LIN {X 0,Y 474.72,Z 465.35,A -85,B 0,C 180,E1 -7388.514,E2 -7388.514} C_VEL
LIN {X 0,Y 474.696,Z 465.35,A -85,B 0,C 180,E1 -7391.963,E2 -7391.963} C_VEL
LIN {X 0,Y 474.691,Z 465.345,A -85,B 0,C 180,E1 -7395.456,E2 -7395.456} C_VEL
LIN {X 0,Y 474.657,Z 465.36,A -85,B 0,C 180,E1 -7399.011,E2 -7399.011} C_VEL
LIN {X 0,Y 474.581,Z 465.36,A -85,B 0,C 180,E1 -7401.729,E2 -7401.729} C_VEL
LIN {X 0,Y 474.651,Z 465.358,A -85,B 0,C 180,E1 -7404.493,E2 -7404.493} C_VEL
LIN {X 0,Y 474.692,Z 465.348,A -85,B 0,C 180,E1 -7407.339,E2 -7407.339} C_VEL
LIN {X 0,Y 474.603,Z 465.346,A -85,B 0,C 180,E1 -7410.812,E2 -7410.812} C_VEL
LIN {X 0,Y 474.632,Z 465.355,A -85,B 0,C 180,E1 -7413.985,E2 -7413.985} C_VEL
LIN {X 0,Y 474.57,Z 465.371,A -85,B 0,C 180,E1 -7416.901,E2 -7416.901} C_VEL
LIN {X 0,Y 474.613,Z 465.345,A -85,B 0,C 180,E1 -7419.647,E2 -7419.647} C_VEL
LIN {X 0,Y 474.627,Z 465.363,A -85,B 0,C 180,E1 -7422.933,E2 -7422.933} C_VEL
LIN {X 0,Y 474.611,Z 465.357,A -85,B 0,C 180,E1 -7425.897,E2 -7425.897} C_VEL
LIN {X 0,Y 474.629,Z 465.361,A -85,B 0,C 180,E1 -7429.041,E2 -7429.041} C_VEL
LIN {X 0,Y 474.613,Z 465.359,A -85,B 0,C 180,E1 -7431.704,E2 -7431.704} C_VEL
LIN {X 0,Y 474.627,Z 465.337,A -85,B 0,C 180,E1 -7434.727,E2 -7434.727} C_VEL
LIN {X 0,Y 474.637,Z 465.356,A -85,B 0,C 180,E1 -7437.789,E2 -7437.789} C_VEL
LIN {X 0,Y 474.624,Z 465.363,A -85,B 0,C 180,E1 -7440.885,E2 -7440.885} C_VEL
LIN {X 0,Y 474.661,Z 465.347,A -85,B 0,C 180,E1 -7443.629,E2 -7443.629} C_VEL
LIN {X 0,Y 474.637,Z 465.361,A -85,B 0,C 180,E1 -7446.642,E2 -7446.642} C_VEL
LIN {X 0,Y 474.659,Z 465.358,A -85,B 0,C 180,E1 -7450.09,E2 -7450.09} C_VEL
LIN {X 0,Y 474.656,Z 465.329,A -85,B 0,C 180,E1 -7451.688,E2 -7451.688} C_VEL
LIN {X 0,Y 474.507,Z 466.016,A -85,B 0,C 180,E1 -7452.131,E2 -7452.131} C_VEL
LIN {X 0,Y 474.153,Z 467.747,A -85,B 0,C 180,E1 -7452.533,E2 -7452.533} C_VEL
LIN {X 0,Y 473.419,Z 471.634,A -85,B 0,C 180,E1 -7453.047,E2 -7453.047} C_VEL
LIN {X 0,Y 472.593,Z 476.648,A -85,B 0,C 180,E1 -7453.451,E2 -7453.451} C_VEL
LIN {X 0,Y 471.86,Z 482.314,A -85,B 0,C 180,E1 -7453.745,E2 -7453.745} C_VEL
LIN {X 0,Y 471.447,Z 488.35,A -85,B 0,C 180,E1 -7453.907,E2 -7453.907} C_VEL
LIN {X 0,Y 471.092,Z 547.467,A -85,B 0,C 180,E1 -7454.839,E2 -7454.839} C_VEL
LIN {X 0,Y 471.01,Z 560.516,A -85,B 0,C 180,E1 -7455.223,E2 -7455.223} C_VEL
LIN {X 0,Y 470.78,Z 572.512,A -85,B 0,C 180,E1 -7455.741,E2 -7455.741} C_VEL
LIN {X 0,Y 470.513,Z 583.759,A -85,B 0,C 180,E1 -7456.392,E2 -7456.392} C_VEL
LIN {X 0,Y 470.007,Z 595.351,A -85,B 0,C 180,E1 -7457.259,E2 -7457.259} C_VEL
LIN {X 0,Y 469.554,Z 605.694,A -85,B 0,C 180,E1 -7458.233,E2 -7458.233} C_VEL
LIN {X 0,Y 469.147,Z 614.13,A -85,B 0,C 180,E1 -7459.208,E2 -7459.208} C_VEL
LIN {X 0,Y 468.818,Z 621.878,A -85,B 0,C 180,E1 -7460.291,E2 -7460.291} C_VEL
LIN {X 0,Y 468.374,Z 629.568,A -85,B 0,C 180,E1 -7461.609,E2 -7461.609} C_VEL
LIN {X 0,Y 468.091,Z 635.326,A -85,B 0,C 180,E1 -7462.84,E2 -7462.84} C_VEL
LIN {X 0,Y 467.937,Z 639.602,A -85,B 0,C 180,E1 -7463.965,E2 -7463.965} C_VEL
LIN {X 0,Y 467.644,Z 643.493,A -85,B 0,C 180,E1 -7465.259,E2 -7465.259} C_VEL
LIN {X 0,Y 467.456,Z 646.362,A -85,B 0,C 180,E1 -7466.552,E2 -7466.552} C_VEL
LIN {X 0,Y 467.483,Z 647.723,A -85,B 0,C 180,E1 -7467.415,E2 -7467.415} C_VEL
LIN {X 0,Y 467.356,Z 648.71,A -85,B 0,C 180,E1 -7468.277,E2 -7468.277} C_VEL
LIN {X 0,Y 467.432,Z 649.296,A -85,B 0,C 180,E1 -7469.139,E2 -7469.139} C_VEL
LIN {X 0,Y 467.416,Z 649.528,A -85,B 0,C 180,E1 -7470,E2 -7470} C_VEL
LIN {X 0,Y 467.432,Z 649.346,A -85,B 0,C 180,E1 -7470.861,E2 -7470.861} C_VEL
LIN {X 0,Y 467.356,Z 648.79,A -85,B 0,C 180,E1 -7471.723,E2 -7471.723} C_VEL
LIN {X 0,Y 467.482,Z 647.836,A -85,B 0,C 180,E1 -7472.585,E2 -7472.585} C_VEL
LIN {X 0,Y 467.451,Z 646.526,A -85,B 0,C 180,E1 -7473.448,E2 -7473.448} C_VEL
LIN {X 0,Y 467.639,Z 643.718,A -85,B 0,C 180,E1 -7474.741,E2 -7474.741} C_VEL
LIN {X 0,Y 467.925,Z 639.903,A -85,B 0,C 180,E1 -7476.035,E2 -7476.035} C_VEL
LIN {X 0,Y 468.063,Z 634.827,A -85,B 0,C 180,E1 -7477.377,E2 -7477.377} C_VEL
LIN {X 0,Y 468.404,Z 628.813,A -85,B 0,C 180,E1 -7478.629,E2 -7478.629} C_VEL
LIN {X 0,Y 468.879,Z 621.039,A -85,B 0,C 180,E1 -7479.926,E2 -7479.926} C_VEL
LIN {X 0,Y 469.297,Z 611.375,A -85,B 0,C 180,E1 -7481.226,E2 -7481.226} C_VEL
LIN {X 0,Y 469.741,Z 602.348,A -85,B 0,C 180,E1 -7482.2,E2 -7482.2} C_VEL
LIN {X 0,Y 470.229,Z 591.863,A -85,B 0,C 180,E1 -7483.114,E2 -7483.114} C_VEL
LIN {X 0,Y 470.571,Z 580.37,A -85,B 0,C 180,E1 -7483.914,E2 -7483.914} C_VEL
LIN {X 0,Y 470.851,Z 569.136,A -85,B 0,C 180,E1 -7484.517,E2 -7484.517} C_VEL
LIN {X 0,Y 471.03,Z 555.98,A -85,B 0,C 180,E1 -7485.025,E2 -7485.025} C_VEL
LIN {X 0,Y 471.055,Z 542.285,A -85,B 0,C 180,E1 -7485.356,E2 -7485.356} C_VEL
LIN {X 0,Y 471.382,Z 476.884,A -85,B 0,C 180,E1 -7486.367,E2 -7486.367} C_VEL
LIN {X 0,Y 467.762,Z 467.093,A -85,B 0,C 180,E1 -7486.689,E2 -7486.689} C_VEL
LIN {X 0,Y 467.626,Z 466.313,A -85,B 0,C 180,E1 -7486.855,E2 -7486.855} C_VEL
LIN {X 0,Y 467.626,Z 466.222,A -85,B 0,C 180,E1 -7489.307,E2 -7489.307} C_VEL
LIN {X 0,Y 467.535,Z 466.233,A -85,B 0,C 180,E1 -7492.073,E2 -7492.073} C_VEL
LIN {X 0,Y 467.604,Z 466.24,A -85,B 0,C 180,E1 -7494.887,E2 -7494.887} C_VEL
LIN {X 0,Y 467.62,Z 466.22,A -85,B 0,C 180,E1 -7497.768,E2 -7497.768} C_VEL
LIN {X 0,Y 467.569,Z 466.243,A -85,B 0,C 180,E1 -7501.044,E2 -7501.044} C_VEL
LIN {X 0,Y 467.588,Z 466.237,A -85,B 0,C 180,E1 -7504.242,E2 -7504.242} C_VEL
LIN {X 0,Y 467.548,Z 466.24,A -85,B 0,C 180,E1 -7507.186,E2 -7507.186} C_VEL
LIN {X 0,Y 467.576,Z 466.239,A -85,B 0,C 180,E1 -7510.264,E2 -7510.264} C_VEL
LIN {X 0,Y 467.583,Z 466.231,A -85,B 0,C 180,E1 -7512.566,E2 -7512.566} C_VEL
LIN {X 0,Y 467.567,Z 466.243,A -85,B 0,C 180,E1 -7515.052,E2 -7515.052} C_VEL
LIN {X 0,Y 467.584,Z 466.237,A -85,B 0,C 180,E1 -7517.439,E2 -7517.439} C_VEL
LIN {X 0,Y 467.555,Z 466.226,A -85,B 0,C 180,E1 -7520.852,E2 -7520.852} C_VEL
LIN {X 0,Y 467.557,Z 466.24,A -85,B 0,C 180,E1 -7524.259,E2 -7524.259} C_VEL
LIN {X 0,Y 467.576,Z 466.229,A -85,B 0,C 180,E1 -7527.32,E2 -7527.32} C_VEL
LIN {X 0,Y 467.571,Z 466.222,A -85,B 0,C 180,E1 -7530.665,E2 -7530.665} C_VEL
LIN {X 0,Y 467.621,Z 466.235,A -85,B 0,C 180,E1 -7533.2,E2 -7533.2} C_VEL
LIN {X 0,Y 467.585,Z 466.234,A -85,B 0,C 180,E1 -7536.468,E2 -7536.468} C_VEL
LIN {X 0,Y 467.615,Z 466.235,A -85,B 0,C 180,E1 -7539.777,E2 -7539.777} C_VEL
LIN {X 0,Y 467.6,Z 466.232,A -85,B 0,C 180,E1 -7542.506,E2 -7542.506} C_VEL
LIN {X 0,Y 467.6,Z 466.235,A -85,B 0,C 180,E1 -7545.196,E2 -7545.196} C_VEL
LIN {X 0,Y 467.647,Z 466.229,A -85,B 0,C 180,E1 -7547.854,E2 -7547.854} C_VEL
LIN {X 0,Y 467.673,Z 466.224,A -85,B 0,C 180,E1 -7551.357,E2 -7551.357} C_VEL
LIN {X 0,Y 467.735,Z 466.218,A -85,B 0,C 180,E1 -7553.962,E2 -7553.962} C_VEL
LIN {X 0,Y 467.851,Z 466.2,A -85,B 0,C 180,E1 -7557.417,E2 -7557.417} C_VEL
LIN {X 0,Y 467.873,Z 466.201,A -85,B 0,C 180,E1 -7560,E2 -7560} C_VEL
LIN {X 0,Y 467.851,Z 466.199,A -85,B 0,C 180,E1 -7562.583,E2 -7562.583} C_VEL
LIN {X 0,Y 467.742,Z 466.217,A -85,B 0,C 180,E1 -7566.037,E2 -7566.037} C_VEL
LIN {X 0,Y 467.673,Z 466.224,A -85,B 0,C 180,E1 -7568.643,E2 -7568.643} C_VEL
LIN {X 0,Y 467.647,Z 466.227,A -85,B 0,C 180,E1 -7572.146,E2 -7572.146} C_VEL
LIN {X 0,Y 467.63,Z 466.233,A -85,B 0,C 180,E1 -7575.695,E2 -7575.695} C_VEL
LIN {X 0,Y 467.608,Z 466.219,A -85,B 0,C 180,E1 -7578.765,E2 -7578.765} C_VEL
LIN {X 0,Y 467.571,Z 466.236,A -85,B 0,C 180,E1 -7581.269,E2 -7581.269} C_VEL
LIN {X 0,Y 467.565,Z 466.241,A -85,B 0,C 180,E1 -7583.944,E2 -7583.944} C_VEL
LIN {X 0,Y 467.619,Z 466.221,A -85,B 0,C 180,E1 -7586.8,E2 -7586.8} C_VEL
LIN {X 0,Y 467.58,Z 466.245,A -85,B 0,C 180,E1 -7589.736,E2 -7589.736} C_VEL
LIN {X 0,Y 467.577,Z 466.231,A -85,B 0,C 180,E1 -7592.759,E2 -7592.759} C_VEL
LIN {X 0,Y 467.551,Z 466.246,A -85,B 0,C 180,E1 -7595.89,E2 -7595.89} C_VEL
LIN {X 0,Y 467.577,Z 466.236,A -85,B 0,C 180,E1 -7599.145,E2 -7599.145} C_VEL
LIN {X 0,Y 467.581,Z 466.23,A -85,B 0,C 180,E1 -7602.568,E2 -7602.568} C_VEL
LIN {X 0,Y 467.566,Z 466.23,A -85,B 0,C 180,E1 -7605.054,E2 -7605.054} C_VEL
LIN {X 0,Y 467.621,Z 466.237,A -85,B 0,C 180,E1 -7607.445,E2 -7607.445} C_VEL
LIN {X 0,Y 467.597,Z 466.235,A -85,B 0,C 180,E1 -7610.858,E2 -7610.858} C_VEL
LIN {X 0,Y 467.56,Z 466.241,A -85,B 0,C 180,E1 -7614.261,E2 -7614.261} C_VEL
LIN {X 0,Y 467.581,Z 466.238,A -85,B 0,C 180,E1 -7617.322,E2 -7617.322} C_VEL
LIN {X 0,Y 467.645,Z 466.452,A -85,B 0,C 180,E1 -7619.663,E2 -7619.663} C_VEL
LIN {X 0,Y 471.182,Z 482.276,A -85,B 0,C 180,E1 -7622.077,E2 -7622.077} C_VEL
LIN {X 0,Y 471.368,Z 486.851,A -85,B 0,C 180,E1 -7622.712,E2 -7622.712} C_VEL
LIN {X 0,Y 470.394,Z 509.213,A -85,B 0,C 180,E1 -7625.697,E2 -7625.697} C_VEL
LIN {X 0,Y 469.471,Z 532.164,A -85,B 0,C 180,E1 -7628.719,E2 -7628.719} C_VEL
LIN {X 0,Y 468.655,Z 556.13,A -85,B 0,C 180,E1 -7631.871,E2 -7631.871} C_VEL
LIN {X 0,Y 468.405,Z 564.473,A -85,B 0,C 180,E1 -7632.944,E2 -7632.944} C_VEL
LIN {X 0,Y 471.027,Z 589.419,A -85,B 0,C 180,E1 -7633.44,E2 -7633.44} C_VEL
LIN {X 0,Y 470.405,Z 674.839,A -85,B 0,C 180,E1 -7634.761,E2 -7634.761} C_VEL
LIN {X 0,Y 470.005,Z 688.179,A -85,B 0,C 180,E1 -7635.136,E2 -7635.136} C_VEL
LIN {X 0,Y 469.551,Z 699.288,A -85,B 0,C 180,E1 -7635.592,E2 -7635.592} C_VEL
LIN {X 0,Y 469.063,Z 711.117,A -85,B 0,C 180,E1 -7636.24,E2 -7636.24} C_VEL
LIN {X 0,Y 468.522,Z 721.919,A -85,B 0,C 180,E1 -7636.997,E2 -7636.997} C_VEL
LIN {X 0,Y 468.141,Z 733.009,A -85,B 0,C 180,E1 -7637.978,E2 -7637.978} C_VEL
LIN {X 0,Y 467.709,Z 742.055,A -85,B 0,C 180,E1 -7638.955,E2 -7638.955} C_VEL
LIN {X 0,Y 467.33,Z 751.917,A -85,B 0,C 180,E1 -7640.26,E2 -7640.26} C_VEL
LIN {X 0,Y 467.117,Z 759.802,A -85,B 0,C 180,E1 -7641.565,E2 -7641.565} C_VEL
LIN {X 0,Y 466.974,Z 767.083,A -85,B 0,C 180,E1 -7643.085,E2 -7643.085} C_VEL
LIN {X 0,Y 466.956,Z 771.946,A -85,B 0,C 180,E1 -7644.386,E2 -7644.386} C_VEL
LIN {X 0,Y 466.96,Z 775.667,A -85,B 0,C 180,E1 -7645.684,E2 -7645.684} C_VEL
LIN {X 0,Y 466.966,Z 777.588,A -85,B 0,C 180,E1 -7646.549,E2 -7646.549} C_VEL
LIN {X 0,Y 466.961,Z 779.029,A -85,B 0,C 180,E1 -7647.412,E2 -7647.412} C_VEL
LIN {X 0,Y 467.06,Z 780.697,A -85,B 0,C 180,E1 -7649.138,E2 -7649.138} C_VEL
LIN {X 0,Y 467.06,Z 780.921,A -85,B 0,C 180,E1 -7650,E2 -7650} C_VEL
LIN {X 0,Y 467.06,Z 780.698,A -85,B 0,C 180,E1 -7650.862,E2 -7650.862} C_VEL
LIN {X 0,Y 466.961,Z 779.032,A -85,B 0,C 180,E1 -7652.588,E2 -7652.588} C_VEL
LIN {X 0,Y 466.966,Z 777.592,A -85,B 0,C 180,E1 -7653.451,E2 -7653.451} C_VEL
LIN {X 0,Y 466.95,Z 774.565,A -85,B 0,C 180,E1 -7654.748,E2 -7654.748} C_VEL
LIN {X 0,Y 466.961,Z 769.403,A -85,B 0,C 180,E1 -7656.332,E2 -7656.332} C_VEL
LIN {X 0,Y 467.021,Z 763.147,A -85,B 0,C 180,E1 -7657.784,E2 -7657.784} C_VEL
LIN {X 0,Y 467.192,Z 756.076,A -85,B 0,C 180,E1 -7659.088,E2 -7659.088} C_VEL
LIN {X 0,Y 467.484,Z 747.251,A -85,B 0,C 180,E1 -7660.393,E2 -7660.393} C_VEL
LIN {X 0,Y 467.803,Z 738.227,A -85,B 0,C 180,E1 -7661.482,E2 -7661.482} C_VEL
LIN {X 0,Y 468.33,Z 728.798,A -85,B 0,C 180,E1 -7662.418,E2 -7662.418} C_VEL
LIN {X 0,Y 468.805,Z 717.598,A -85,B 0,C 180,E1 -7663.326,E2 -7663.326} C_VEL
LIN {X 0,Y 469.283,Z 705.591,A -85,B 0,C 180,E1 -7664.085,E2 -7664.085} C_VEL
LIN {X 0,Y 469.785,Z 693.147,A -85,B 0,C 180,E1 -7664.678,E2 -7664.678} C_VEL
LIN {X 0,Y 470.251,Z 680.413,A -85,B 0,C 180,E1 -7665.106,E2 -7665.106} C_VEL
LIN {X 0,Y 470.489,Z 667.134,A -85,B 0,C 180,E1 -7665.375,E2 -7665.375} C_VEL
LIN {X 0,Y 470.921,Z 587.375,A -85,B 0,C 180,E1 -7666.595,E2 -7666.595} C_VEL
LIN {X 0,Y 468.416,Z 564.827,A -85,B 0,C 180,E1 -7667.04,E2 -7667.04} C_VEL
LIN {X 0,Y 468.449,Z 562.893,A -85,B 0,C 180,E1 -7667.235,E2 -7667.235} C_VEL
LIN {X 0,Y 469.217,Z 539.002,A -85,B 0,C 180,E1 -7670.379,E2 -7670.379} C_VEL
LIN {X 0,Y 469.968,Z 519.985,A -85,B 0,C 180,E1 -7672.88,E2 -7672.88} C_VEL
LIN {X 0,Y 470.929,Z 495.825,A -85,B 0,C 180,E1 -7676.082,E2 -7676.082} C_VEL
LIN {X 0,Y 471.402,Z 483.677,A -85,B 0,C 180,E1 -7677.717,E2 -7677.717} C_VEL
LIN {X 0,Y 468.197,Z 468.878,A -85,B 0,C 180,E1 -7679.94,E2 -7679.94} C_VEL
LIN {X 0,Y 467.602,Z 466.335,A -85,B 0,C 180,E1 -7680.387,E2 -7680.387} C_VEL
LIN {X 0,Y 467.584,Z 466.236,A -85,B 0,C 180,E1 -7683.787,E2 -7683.787} C_VEL
LIN {X 0,Y 467.545,Z 466.24,A -85,B 0,C 180,E1 -7687.186,E2 -7687.186} C_VEL
LIN {X 0,Y 467.593,Z 466.23,A -85,B 0,C 180,E1 -7690.262,E2 -7690.262} C_VEL
LIN {X 0,Y 467.615,Z 466.238,A -85,B 0,C 180,E1 -7692.571,E2 -7692.571} C_VEL
LIN {X 0,Y 467.566,Z 466.23,A -85,B 0,C 180,E1 -7695.052,E2 -7695.052} C_VEL
LIN {X 0,Y 467.584,Z 466.229,A -85,B 0,C 180,E1 -7697.439,E2 -7697.439} C_VEL
LIN {X 0,Y 467.577,Z 466.235,A -85,B 0,C 180,E1 -7700.855,E2 -7700.855} C_VEL
LIN {X 0,Y 467.557,Z 466.248,A -85,B 0,C 180,E1 -7704.26,E2 -7704.26} C_VEL
LIN {X 0,Y 467.576,Z 466.232,A -85,B 0,C 180,E1 -7707.32,E2 -7707.32} C_VEL
LIN {X 0,Y 467.571,Z 466.24,A -85,B 0,C 180,E1 -7710.665,E2 -7710.665} C_VEL
LIN {X 0,Y 467.619,Z 466.222,A -85,B 0,C 180,E1 -7713.2,E2 -7713.2} C_VEL
LIN {X 0,Y 467.584,Z 466.244,A -85,B 0,C 180,E1 -7716.468,E2 -7716.468} C_VEL
LIN {X 0,Y 467.615,Z 466.227,A -85,B 0,C 180,E1 -7719.777,E2 -7719.777} C_VEL
LIN {X 0,Y 467.6,Z 466.23,A -85,B 0,C 180,E1 -7722.506,E2 -7722.506} C_VEL
LIN {X 0,Y 467.596,Z 466.236,A -85,B 0,C 180,E1 -7725.196,E2 -7725.196} C_VEL
LIN {X 0,Y 467.647,Z 466.227,A -85,B 0,C 180,E1 -7727.854,E2 -7727.854} C_VEL
LIN {X 0,Y 467.673,Z 466.225,A -85,B 0,C 180,E1 -7731.357,E2 -7731.357} C_VEL
LIN {X 0,Y 467.743,Z 466.217,A -85,B 0,C 180,E1 -7733.963,E2 -7733.963} C_VEL
LIN {X 0,Y 467.851,Z 466.201,A -85,B 0,C 180,E1 -7737.417,E2 -7737.417} C_VEL
LIN {X 0,Y 467.873,Z 466.202,A -85,B 0,C 180,E1 -7740,E2 -7740} C_VEL
LIN {X 0,Y 467.851,Z 466.201,A -85,B 0,C 180,E1 -7742.583,E2 -7742.583} C_VEL
LIN {X 0,Y 467.744,Z 466.217,A -85,B 0,C 180,E1 -7746.037,E2 -7746.037} C_VEL
LIN {X 0,Y 467.673,Z 466.225,A -85,B 0,C 180,E1 -7748.643,E2 -7748.643} C_VEL
LIN {X 0,Y 467.647,Z 466.229,A -85,B 0,C 180,E1 -7752.146,E2 -7752.146} C_VEL
LIN {X 0,Y 467.63,Z 466.224,A -85,B 0,C 180,E1 -7755.695,E2 -7755.695} C_VEL
LIN {X 0,Y 467.609,Z 466.24,A -85,B 0,C 180,E1 -7758.765,E2 -7758.765} C_VEL
LIN {X 0,Y 467.572,Z 466.235,A -85,B 0,C 180,E1 -7761.269,E2 -7761.269} C_VEL
LIN {X 0,Y 467.565,Z 466.237,A -85,B 0,C 180,E1 -7763.944,E2 -7763.944} C_VEL
LIN {X 0,Y 467.621,Z 466.236,A -85,B 0,C 180,E1 -7766.8,E2 -7766.8} C_VEL
LIN {X 0,Y 467.58,Z 466.219,A -85,B 0,C 180,E1 -7769.736,E2 -7769.736} C_VEL
LIN {X 0,Y 467.577,Z 466.229,A -85,B 0,C 180,E1 -7772.759,E2 -7772.759} C_VEL
LIN {X 0,Y 467.551,Z 466.241,A -85,B 0,C 180,E1 -7775.89,E2 -7775.89} C_VEL
LIN {X 0,Y 467.555,Z 466.228,A -85,B 0,C 180,E1 -7779.148,E2 -7779.148} C_VEL
LIN {X 0,Y 467.582,Z 466.235,A -85,B 0,C 180,E1 -7782.568,E2 -7782.568} C_VEL
LIN {X 0,Y 467.567,Z 466.242,A -85,B 0,C 180,E1 -7785.054,E2 -7785.054} C_VEL
LIN {X 0,Y 467.585,Z 466.229,A -85,B 0,C 180,E1 -7787.441,E2 -7787.441} C_VEL
LIN {X 0,Y 467.583,Z 466.244,A -85,B 0,C 180,E1 -7790.856,E2 -7790.856} C_VEL
LIN {X 0,Y 467.56,Z 466.222,A -85,B 0,C 180,E1 -7794.261,E2 -7794.261} C_VEL
LIN {X 0,Y 467.582,Z 466.227,A -85,B 0,C 180,E1 -7797.322,E2 -7797.322} C_VEL
LIN {X 0,Y 467.57,Z 466.244,A -85,B 0,C 180,E1 -7800.668,E2 -7800.668} C_VEL
LIN {X 0,Y 467.616,Z 466.219,A -85,B 0,C 180,E1 -7803.2,E2 -7803.2} C_VEL
LIN {X 0,Y 467.594,Z 466.238,A -85,B 0,C 180,E1 -7806.469,E2 -7806.469} C_VEL
LIN {X 0,Y 467.626,Z 466.236,A -85,B 0,C 180,E1 -7809.778,E2 -7809.778} C_VEL
LIN {X 0,Y 467.617,Z 466.189,A -85,B 0,C 180,E1 -7812.958,E2 -7812.958} C_VEL
LIN {X 0,Y 467.689,Z 466.544,A -85,B 0,C 180,E1 -7813.327,E2 -7813.327} C_VEL
LIN {X 0,Y 467.986,Z 467.754,A -85,B 0,C 180,E1 -7813.446,E2 -7813.446} C_VEL
LIN {X 0,Y 471.541,Z 477.483,A -85,B 0,C 180,E1 -7813.741,E2 -7813.741} C_VEL
LIN {X 0,Y 471.447,Z 488.35,A -85,B 0,C 180,E1 -7813.907,E2 -7813.907} C_VEL
LIN {X 0,Y 470.68,Z 494.195,A -85,B 0,C 180,E1 -7813.97,E2 -7813.97} C_VEL
LIN {X 0,Y 465.061,Z 513.201,A -85,B 0,C 180,E1 -7814.058,E2 -7814.058} C_VEL
LIN {X 0,Y 464.429,Z 519.041,A -85,B 0,C 180,E1 -7814.127,E2 -7814.127} C_VEL
LIN {X 0,Y 464.29,Z 548.477,A -85,B 0,C 180,E1 -7814.611,E2 -7814.611} C_VEL
LIN {X 0,Y 464.209,Z 561.518,A -85,B 0,C 180,E1 -7815.002,E2 -7815.002} C_VEL
LIN {X 0,Y 463.968,Z 573.509,A -85,B 0,C 180,E1 -7815.527,E2 -7815.527} C_VEL
LIN {X 0,Y 463.686,Z 584.754,A -85,B 0,C 180,E1 -7816.188,E2 -7816.188} C_VEL
LIN {X 0,Y 463.153,Z 596.345,A -85,B 0,C 180,E1 -7817.067,E2 -7817.067} C_VEL
LIN {X 0,Y 462.675,Z 606.686,A -85,B 0,C 180,E1 -7818.056,E2 -7818.056} C_VEL
LIN {X 0,Y 462.246,Z 615.122,A -85,B 0,C 180,E1 -7819.045,E2 -7819.045} C_VEL
LIN {X 0,Y 461.893,Z 622.869,A -85,B 0,C 180,E1 -7820.144,E2 -7820.144} C_VEL
LIN {X 0,Y 461.423,Z 630.558,A -85,B 0,C 180,E1 -7821.482,E2 -7821.482} C_VEL
LIN {X 0,Y 461.119,Z 636.316,A -85,B 0,C 180,E1 -7822.732,E2 -7822.732} C_VEL
LIN {X 0,Y 460.953,Z 640.591,A -85,B 0,C 180,E1 -7823.873,E2 -7823.873} C_VEL
LIN {X 0,Y 460.638,Z 644.483,A -85,B 0,C 180,E1 -7825.187,E2 -7825.187} C_VEL
LIN {X 0,Y 460.438,Z 647.351,A -85,B 0,C 180,E1 -7826.5,E2 -7826.5} C_VEL
LIN {X 0,Y 460.466,Z 648.711,A -85,B 0,C 180,E1 -7827.376,E2 -7827.376} C_VEL
LIN {X 0,Y 460.334,Z 649.698,A -85,B 0,C 180,E1 -7828.25,E2 -7828.25} C_VEL
LIN {X 0,Y 460.412,Z 650.284,A -85,B 0,C 180,E1 -7829.125,E2 -7829.125} C_VEL
LIN {X 0,Y 460.396,Z 650.516,A -85,B 0,C 180,E1 -7830,E2 -7830} C_VEL
LIN {X 0,Y 460.412,Z 650.333,A -85,B 0,C 180,E1 -7830.875,E2 -7830.875} C_VEL
LIN {X 0,Y 460.334,Z 649.778,A -85,B 0,C 180,E1 -7831.75,E2 -7831.75} C_VEL
LIN {X 0,Y 460.465,Z 648.823,A -85,B 0,C 180,E1 -7832.624,E2 -7832.624} C_VEL
LIN {X 0,Y 460.433,Z 647.514,A -85,B 0,C 180,E1 -7833.5,E2 -7833.5} C_VEL
LIN {X 0,Y 460.632,Z 644.706,A -85,B 0,C 180,E1 -7834.814,E2 -7834.814} C_VEL
LIN {X 0,Y 460.939,Z 640.889,A -85,B 0,C 180,E1 -7836.127,E2 -7836.127} C_VEL
LIN {X 0,Y 461.094,Z 635.814,A -85,B 0,C 180,E1 -7837.488,E2 -7837.488} C_VEL
LIN {X 0,Y 461.459,Z 629.798,A -85,B 0,C 180,E1 -7838.76,E2 -7838.76} C_VEL
LIN {X 0,Y 461.959,Z 622.024,A -85,B 0,C 180,E1 -7840.076,E2 -7840.076} C_VEL
LIN {X 0,Y 462.404,Z 612.36,A -85,B 0,C 180,E1 -7841.395,E2 -7841.395} C_VEL
LIN {X 0,Y 462.872,Z 603.332,A -85,B 0,C 180,E1 -7842.384,E2 -7842.384} C_VEL
LIN {X 0,Y 463.387,Z 592.845,A -85,B 0,C 180,E1 -7843.311,E2 -7843.311} C_VEL
LIN {X 0,Y 463.752,Z 581.351,A -85,B 0,C 180,E1 -7844.123,E2 -7844.123} C_VEL
LIN {X 0,Y 464.047,Z 570.116,A -85,B 0,C 180,E1 -7844.734,E2 -7844.734} C_VEL
LIN {X 0,Y 464.23,Z 556.956,A -85,B 0,C 180,E1 -7845.25,E2 -7845.25} C_VEL
LIN {X 0,Y 464.246,Z 543.254,A -85,B 0,C 180,E1 -7845.587,E2 -7845.587} C_VEL
LIN {X 0,Y 464.671,Z 478.577,A -85,B 0,C 180,E1 -7846.599,E2 -7846.599} C_VEL
LIN {X 0,Y 460.774,Z 468.175,A -85,B 0,C 180,E1 -7846.936,E2 -7846.936} C_VEL
LIN {X 0,Y 460.623,Z 467.265,A -85,B 0,C 180,E1 -7847.08,E2 -7847.08} C_VEL
LIN {X 0,Y 460.572,Z 467.108,A -85,B 0,C 180,E1 -7849.615,E2 -7849.615} C_VEL
LIN {X 0,Y 460.512,Z 467.107,A -85,B 0,C 180,E1 -7852.428,E2 -7852.428} C_VEL
LIN {X 0,Y 460.568,Z 467.107,A -85,B 0,C 180,E1 -7855.801,E2 -7855.801} C_VEL
LIN {X 0,Y 460.552,Z 467.101,A -85,B 0,C 180,E1 -7858.232,E2 -7858.232} C_VEL
LIN {X 0,Y 460.521,Z 467.118,A -85,B 0,C 180,E1 -7861.282,E2 -7861.282} C_VEL
LIN {X 0,Y 460.532,Z 467.118,A -85,B 0,C 180,E1 -7864.505,E2 -7864.505} C_VEL
LIN {X 0,Y 460.526,Z 467.115,A -85,B 0,C 180,E1 -7867.62,E2 -7867.62} C_VEL
LIN {X 0,Y 460.54,Z 467.115,A -85,B 0,C 180,E1 -7870.269,E2 -7870.269} C_VEL
LIN {X 0,Y 460.505,Z 467.115,A -85,B 0,C 180,E1 -7873.373,E2 -7873.373} C_VEL
LIN {X 0,Y 460.496,Z 467.123,A -85,B 0,C 180,E1 -7876.624,E2 -7876.624} C_VEL
LIN {X 0,Y 460.534,Z 467.096,A -85,B 0,C 180,E1 -7879.73,E2 -7879.73} C_VEL
LIN {X 0,Y 460.522,Z 467.113,A -85,B 0,C 180,E1 -7882.519,E2 -7882.519} C_VEL
LIN {X 0,Y 460.543,Z 467.113,A -85,B 0,C 180,E1 -7885.623,E2 -7885.623} C_VEL
LIN {X 0,Y 460.53,Z 467.099,A -85,B 0,C 180,E1 -7888.744,E2 -7888.744} C_VEL
LIN {X 0,Y 460.551,Z 467.109,A -85,B 0,C 180,E1 -7891.767,E2 -7891.767} C_VEL
LIN {X 0,Y 460.552,Z 467.114,A -85,B 0,C 180,E1 -7894.705,E2 -7894.705} C_VEL
LIN {X 0,Y 460.503,Z 467.117,A -85,B 0,C 180,E1 -7897.571,E2 -7897.571} C_VEL
LIN {X 0,Y 460.561,Z 467.111,A -85,B 0,C 180,E1 -7900.384,E2 -7900.384} C_VEL
LIN {X 0,Y 460.557,Z 467.113,A -85,B 0,C 180,E1 -7903.146,E2 -7903.146} C_VEL
LIN {X 0,Y 460.548,Z 467.114,A -85,B 0,C 180,E1 -7905.868,E2 -7905.868} C_VEL
LIN {X 0,Y 460.604,Z 467.105,A -85,B 0,C 180,E1 -7908.559,E2 -7908.559} C_VEL
LIN {X 0,Y 460.686,Z 467.093,A -85,B 0,C 180,E1 -7912.108,E2 -7912.108} C_VEL
LIN {X 0,Y 460.689,Z 467.095,A -85,B 0,C 180,E1 -7914.748,E2 -7914.748} C_VEL
LIN {X 0,Y 460.816,Z 467.076,A -85,B 0,C 180,E1 -7917.378,E2 -7917.378} C_VEL
LIN {X 0,Y 460.844,Z 467.076,A -85,B 0,C 180,E1 -7920,E2 -7920} C_VEL
LIN {X 0,Y 460.816,Z 467.076,A -85,B 0,C 180,E1 -7922.622,E2 -7922.622} C_VEL
LIN {X 0,Y 460.707,Z 467.093,A -85,B 0,C 180,E1 -7926.13,E2 -7926.13} C_VEL
LIN {X 0,Y 460.62,Z 467.103,A -85,B 0,C 180,E1 -7928.776,E2 -7928.776} C_VEL
LIN {X 0,Y 460.604,Z 467.103,A -85,B 0,C 180,E1 -7932.445,E2 -7932.445} C_VEL
LIN {X 0,Y 460.591,Z 467.106,A -85,B 0,C 180,E1 -7935.998,E2 -7935.998} C_VEL
LIN {X 0,Y 460.562,Z 467.096,A -85,B 0,C 180,E1 -7938.902,E2 -7938.902} C_VEL
LIN {X 0,Y 460.507,Z 467.119,A -85,B 0,C 180,E1 -7941.486,E2 -7941.486} C_VEL
LIN {X 0,Y 460.534,Z 467.114,A -85,B 0,C 180,E1 -7944.333,E2 -7944.333} C_VEL
LIN {X 0,Y 460.576,Z 467.101,A -85,B 0,C 180,E1 -7947.244,E2 -7947.244} C_VEL
LIN {X 0,Y 460.52,Z 467.118,A -85,B 0,C 180,E1 -7950.239,E2 -7950.239} C_VEL
LIN {X 0,Y 460.523,Z 467.112,A -85,B 0,C 180,E1 -7953.325,E2 -7953.325} C_VEL
LIN {X 0,Y 460.473,Z 467.122,A -85,B 0,C 180,E1 -7956.53,E2 -7956.53} C_VEL
LIN {X 0,Y 460.552,Z 467.12,A -85,B 0,C 180,E1 -7959.86,E2 -7959.86} C_VEL
LIN {X 0,Y 460.508,Z 467.11,A -85,B 0,C 180,E1 -7962.901,E2 -7962.901} C_VEL
LIN {X 0,Y 460.52,Z 467.116,A -85,B 0,C 180,E1 -7965.83,E2 -7965.83} C_VEL
LIN {X 0,Y 460.54,Z 467.11,A -85,B 0,C 180,E1 -7968.991,E2 -7968.991} C_VEL
LIN {X 0,Y 460.537,Z 467.116,A -85,B 0,C 180,E1 -7971.269,E2 -7971.269} C_VEL
LIN {X 0,Y 460.511,Z 467.122,A -85,B 0,C 180,E1 -7974.555,E2 -7974.555} C_VEL
LIN {X 0,Y 460.531,Z 467.121,A -85,B 0,C 180,E1 -7977.716,E2 -7977.716} C_VEL
LIN {X 0,Y 460.557,Z 467.27,A -85,B 0,C 180,E1 -7979.384,E2 -7979.384} C_VEL
LIN {X 0,Y 463.671,Z 480.972,A -85,B 0,C 180,E1 -7981.537,E2 -7981.537} C_VEL
LIN {X 0,Y 464.523,Z 485.958,A -85,B 0,C 180,E1 -7982.275,E2 -7982.275} C_VEL
LIN {X 0,Y 463.556,Z 507.795,A -85,B 0,C 180,E1 -7985.246,E2 -7985.246} C_VEL
LIN {X 0,Y 462.605,Z 530.098,A -85,B 0,C 180,E1 -7988.236,E2 -7988.236} C_VEL
LIN {X 0,Y 461.714,Z 553.447,A -85,B 0,C 180,E1 -7991.359,E2 -7991.359} C_VEL
LIN {X 0,Y 461.41,Z 563.471,A -85,B 0,C 180,E1 -7992.677,E2 -7992.677} C_VEL
LIN {X 0,Y 464.186,Z 590.414,A -85,B 0,C 180,E1 -7993.22,E2 -7993.22} C_VEL
LIN {X 0,Y 463.527,Z 673.845,A -85,B 0,C 180,E1 -7994.529,E2 -7994.529} C_VEL
LIN {X 0,Y 463.113,Z 687.182,A -85,B 0,C 180,E1 -7994.909,E2 -7994.909} C_VEL
LIN {X 0,Y 462.617,Z 698.285,A -85,B 0,C 180,E1 -7995.371,E2 -7995.371} C_VEL
LIN {X 0,Y 462.092,Z 710.11,A -85,B 0,C 180,E1 -7996.029,E2 -7996.029} C_VEL
LIN {X 0,Y 461.506,Z 721.979,A -85,B 0,C 180,E1 -7996.885,E2 -7996.885} C_VEL
LIN {X 0,Y 461.089,Z 733.092,A -85,B 0,C 180,E1 -7997.903,E2 -7997.903} C_VEL
LIN {X 0,Y 460.584,Z 742.865,A -85,B 0,C 180,E1 -7999.005,E2 -7999.005} C_VEL
LIN {X 0,Y 460.273,Z 750.911,A -85,B 0,C 180,E1 -8000.109,E2 -8000.109} C_VEL
LIN {X 0,Y 460.034,Z 758.795,A -85,B 0,C 180,E1 -8001.434,E2 -8001.434} C_VEL
LIN {X 0,Y 459.92,Z 766.085,A -85,B 0,C 180,E1 -8002.978,E2 -8002.978} C_VEL
LIN {X 0,Y 459.899,Z 770.949,A -85,B 0,C 180,E1 -8004.3,E2 -8004.3} C_VEL
LIN {X 0,Y 459.907,Z 774.673,A -85,B 0,C 180,E1 -8005.618,E2 -8005.618} C_VEL
LIN {X 0,Y 459.921,Z 776.596,A -85,B 0,C 180,E1 -8006.496,E2 -8006.496} C_VEL
LIN {X 0,Y 459.916,Z 778.037,A -85,B 0,C 180,E1 -8007.373,E2 -8007.373} C_VEL
LIN {X 0,Y 460.042,Z 779.711,A -85,B 0,C 180,E1 -8009.125,E2 -8009.125} C_VEL
LIN {X 0,Y 460.043,Z 779.934,A -85,B 0,C 180,E1 -8010,E2 -8010} C_VEL
LIN {X 0,Y 460.042,Z 779.711,A -85,B 0,C 180,E1 -8010.875,E2 -8010.875} C_VEL
LIN {X 0,Y 459.916,Z 778.041,A -85,B 0,C 180,E1 -8012.627,E2 -8012.627} C_VEL
LIN {X 0,Y 459.921,Z 776.6,A -85,B 0,C 180,E1 -8013.504,E2 -8013.504} C_VEL
LIN {X 0,Y 459.903,Z 773.57,A -85,B 0,C 180,E1 -8014.821,E2 -8014.821} C_VEL
LIN {X 0,Y 459.91,Z 769.475,A -85,B 0,C 180,E1 -8016.14,E2 -8016.14} C_VEL
LIN {X 0,Y 459.942,Z 763.183,A -85,B 0,C 180,E1 -8017.683,E2 -8017.683} C_VEL
LIN {X 0,Y 460.08,Z 756.333,A -85,B 0,C 180,E1 -8019.008,E2 -8019.008} C_VEL
LIN {X 0,Y 460.366,Z 747.864,A -85,B 0,C 180,E1 -8020.333,E2 -8020.333} C_VEL
LIN {X 0,Y 460.701,Z 739.203,A -85,B 0,C 180,E1 -8021.438,E2 -8021.438} C_VEL
LIN {X 0,Y 461.29,Z 728.384,A -85,B 0,C 180,E1 -8022.555,E2 -8022.555} C_VEL
LIN {X 0,Y 461.801,Z 716.583,A -85,B 0,C 180,E1 -8023.532,E2 -8023.532} C_VEL
LIN {X 0,Y 462.39,Z 704.588,A -85,B 0,C 180,E1 -8024.299,E2 -8024.299} C_VEL
LIN {X 0,Y 462.873,Z 692.137,A -85,B 0,C 180,E1 -8024.902,E2 -8024.902} C_VEL
LIN {X 0,Y 463.397,Z 679.407,A -85,B 0,C 180,E1 -8025.335,E2 -8025.335} C_VEL
LIN {X 0,Y 463.647,Z 666.121,A -85,B 0,C 180,E1 -8025.608,E2 -8025.608} C_VEL
LIN {X 0,Y 464.058,Z 587.589,A -85,B 0,C 180,E1 -8026.828,E2 -8026.828} C_VEL
LIN {X 0,Y 461.406,Z 563.462,A -85,B 0,C 180,E1 -8027.322,E2 -8027.322} C_VEL
LIN {X 0,Y 462.29,Z 538.039,A -85,B 0,C 180,E1 -8030.699,E2 -8030.699} C_VEL
LIN {X 0,Y 463.007,Z 519.039,A -85,B 0,C 180,E1 -8033.244,E2 -8033.244} C_VEL
LIN {X 0,Y 463.95,Z 498.139,A -85,B 0,C 180,E1 -8036.058,E2 -8036.058} C_VEL
LIN {X 0,Y 464.526,Z 485.926,A -85,B 0,C 180,E1 -8037.724,E2 -8037.724} C_VEL
LIN {X 0,Y 462.234,Z 474.17,A -85,B 0,C 180,E1 -8039.497,E2 -8039.497} C_VEL
LIN {X 0,Y 460.577,Z 467.229,A -85,B 0,C 180,E1 -8040.63,E2 -8040.63} C_VEL
LIN {X 0,Y 460.527,Z 467.113,A -85,B 0,C 180,E1 -8043.324,E2 -8043.324} C_VEL
LIN {X 0,Y 460.474,Z 467.12,A -85,B 0,C 180,E1 -8046.529,E2 -8046.529} C_VEL
LIN {X 0,Y 460.572,Z 467.106,A -85,B 0,C 180,E1 -8049.857,E2 -8049.857} C_VEL
LIN {X 0,Y 460.539,Z 467.117,A -85,B 0,C 180,E1 -8052.904,E2 -8052.904} C_VEL
LIN {X 0,Y 460.507,Z 467.105,A -85,B 0,C 180,E1 -8055.83,E2 -8055.83} C_VEL
LIN {X 0,Y 460.526,Z 467.117,A -85,B 0,C 180,E1 -8058.988,E2 -8058.988} C_VEL
LIN {X 0,Y 460.521,Z 467.113,A -85,B 0,C 180,E1 -8061.266,E2 -8061.266} C_VEL
LIN {X 0,Y 460.507,Z 467.122,A -85,B 0,C 180,E1 -8064.554,E2 -8064.554} C_VEL
LIN {X 0,Y 460.526,Z 467.111,A -85,B 0,C 180,E1 -8067.715,E2 -8067.715} C_VEL
LIN {X 0,Y 460.54,Z 467.114,A -85,B 0,C 180,E1 -8070.769,E2 -8070.769} C_VEL
LIN {X 0,Y 460.56,Z 467.101,A -85,B 0,C 180,E1 -8073.734,E2 -8073.734} C_VEL
LIN {X 0,Y 460.538,Z 467.119,A -85,B 0,C 180,E1 -8076.623,E2 -8076.623} C_VEL
LIN {X 0,Y 460.543,Z 467.107,A -85,B 0,C 180,E1 -8079.452,E2 -8079.452} C_VEL
LIN {X 0,Y 460.55,Z 467.103,A -85,B 0,C 180,E1 -8082.23,E2 -8082.23} C_VEL
LIN {X 0,Y 460.555,Z 467.114,A -85,B 0,C 180,E1 -8084.965,E2 -8084.965} C_VEL
LIN {X 0,Y 460.604,Z 467.104,A -85,B 0,C 180,E1 -8088.559,E2 -8088.559} C_VEL
LIN {X 0,Y 460.685,Z 467.098,A -85,B 0,C 180,E1 -8092.108,E2 -8092.108} C_VEL
LIN {X 0,Y 460.696,Z 467.091,A -85,B 0,C 180,E1 -8094.748,E2 -8094.748} C_VEL
LIN {X 0,Y 460.816,Z 467.078,A -85,B 0,C 180,E1 -8097.378,E2 -8097.378} C_VEL
LIN {X 0,Y 460.844,Z 467.077,A -85,B 0,C 180,E1 -8100,E2 -8100} C_VEL
LIN {X 0,Y 460.816,Z 467.077,A -85,B 0,C 180,E1 -8102.622,E2 -8102.622} C_VEL
LIN {X 0,Y 460.709,Z 467.094,A -85,B 0,C 180,E1 -8106.13,E2 -8106.13} C_VEL
LIN {X 0,Y 460.62,Z 467.101,A -85,B 0,C 180,E1 -8108.776,E2 -8108.776} C_VEL
LIN {X 0,Y 460.604,Z 467.109,A -85,B 0,C 180,E1 -8112.445,E2 -8112.445} C_VEL
LIN {X 0,Y 460.591,Z 467.101,A -85,B 0,C 180,E1 -8115.998,E2 -8115.998} C_VEL
LIN {X 0,Y 460.563,Z 467.117,A -85,B 0,C 180,E1 -8118.902,E2 -8118.902} C_VEL
LIN {X 0,Y 460.508,Z 467.114,A -85,B 0,C 180,E1 -8121.486,E2 -8121.486} C_VEL
LIN {X 0,Y 460.535,Z 467.115,A -85,B 0,C 180,E1 -8124.333,E2 -8124.333} C_VEL
LIN {X 0,Y 460.577,Z 467.107,A -85,B 0,C 180,E1 -8127.244,E2 -8127.244} C_VEL
LIN {X 0,Y 460.52,Z 467.099,A -85,B 0,C 180,E1 -8130.24,E2 -8130.24} C_VEL
LIN {X 0,Y 460.523,Z 467.115,A -85,B 0,C 180,E1 -8133.326,E2 -8133.326} C_VEL
LIN {X 0,Y 460.473,Z 467.126,A -85,B 0,C 180,E1 -8136.53,E2 -8136.53} C_VEL
LIN {X 0,Y 460.529,Z 467.106,A -85,B 0,C 180,E1 -8138.897,E2 -8138.897} C_VEL
LIN {X 0,Y 460.518,Z 467.112,A -85,B 0,C 180,E1 -8142.182,E2 -8142.182} C_VEL
LIN {X 0,Y 460.516,Z 467.115,A -85,B 0,C 180,E1 -8145.413,E2 -8145.413} C_VEL
LIN {X 0,Y 460.532,Z 467.108,A -85,B 0,C 180,E1 -8148.398,E2 -8148.398} C_VEL
LIN {X 0,Y 460.53,Z 467.117,A -85,B 0,C 180,E1 -8151.268,E2 -8151.268} C_VEL
LIN {X 0,Y 460.511,Z 467.094,A -85,B 0,C 180,E1 -8154.555,E2 -8154.555} C_VEL
LIN {X 0,Y 460.532,Z 467.114,A -85,B 0,C 180,E1 -8157.717,E2 -8157.717} C_VEL
LIN {X 0,Y 460.54,Z 467.119,A -85,B 0,C 180,E1 -8160.77,E2 -8160.77} C_VEL
LIN {X 0,Y 460.563,Z 467.102,A -85,B 0,C 180,E1 -8163.735,E2 -8163.735} C_VEL
LIN {X 0,Y 460.547,Z 467.114,A -85,B 0,C 180,E1 -8166.625,E2 -8166.625} C_VEL
LIN {X 0,Y 460.555,Z 467.12,A -85,B 0,C 180,E1 -8169.453,E2 -8169.453} C_VEL
LIN {X 0,Y 460.559,Z 467.07,A -85,B 0,C 180,E1 -8172.231,E2 -8172.231} C_VEL
LIN {X 0,Y 460.628,Z 467.325,A -85,B 0,C 180,E1 -8173.035,E2 -8173.035} C_VEL
LIN {X 0,Y 460.819,Z 468.23,A -85,B 0,C 180,E1 -8173.162,E2 -8173.162} C_VEL
LIN {X 0,Y 464.736,Z 479.2,A -85,B 0,C 180,E1 -8173.508,E2 -8173.508} C_VEL
LIN {X 0,Y 464.429,Z 519.041,A -85,B 0,C 180,E1 -8174.127,E2 -8174.127} C_VEL
LIN {X 0,Y 463.777,Z 524.896,A -85,B 0,C 180,E1 -8174.19,E2 -8174.19} C_VEL
LIN {X 0,Y 458.149,Z 543.91,A -85,B 0,C 180,E1 -8174.276,E2 -8174.276} C_VEL
LIN {X 0,Y 457.51,Z 549.705,A -85,B 0,C 180,E1 -8174.383,E2 -8174.383} C_VEL
LIN {X 0,Y 457.394,Z 563.275,A -85,B 0,C 180,E1 -8174.801,E2 -8174.801} C_VEL
LIN {X 0,Y 457.154,Z 575.709,A -85,B 0,C 180,E1 -8175.369,E2 -8175.369} C_VEL
LIN {X 0,Y 456.796,Z 586.937,A -85,B 0,C 180,E1 -8176.06,E2 -8176.06} C_VEL
LIN {X 0,Y 456.244,Z 598.609,A -85,B 0,C 180,E1 -8176.981,E2 -8176.981} C_VEL
LIN {X 0,Y 455.753,Z 608.726,A -85,B 0,C 180,E1 -8177.985,E2 -8177.985} C_VEL
LIN {X 0,Y 455.284,Z 617.786,A -85,B 0,C 180,E1 -8179.1,E2 -8179.1} C_VEL
LIN {X 0,Y 454.795,Z 626.558,A -85,B 0,C 180,E1 -8180.438,E2 -8180.438} C_VEL
LIN {X 0,Y 454.406,Z 632.744,A -85,B 0,C 180,E1 -8181.596,E2 -8181.596} C_VEL
LIN {X 0,Y 454.119,Z 638.361,A -85,B 0,C 180,E1 -8182.888,E2 -8182.888} C_VEL
LIN {X 0,Y 453.766,Z 642.985,A -85,B 0,C 180,E1 -8184.222,E2 -8184.222} C_VEL
LIN {X 0,Y 453.544,Z 646.515,A -85,B 0,C 180,E1 -8185.556,E2 -8185.556} C_VEL
LIN {X 0,Y 453.421,Z 648.341,A -85,B 0,C 180,E1 -8186.445,E2 -8186.445} C_VEL
LIN {X 0,Y 453.449,Z 649.7,A -85,B 0,C 180,E1 -8187.335,E2 -8187.335} C_VEL
LIN {X 0,Y 453.313,Z 650.686,A -85,B 0,C 180,E1 -8188.223,E2 -8188.223} C_VEL
LIN {X 0,Y 453.391,Z 651.271,A -85,B 0,C 180,E1 -8189.112,E2 -8189.112} C_VEL
LIN {X 0,Y 453.375,Z 651.503,A -85,B 0,C 180,E1 -8190,E2 -8190} C_VEL
LIN {X 0,Y 453.391,Z 651.32,A -85,B 0,C 180,E1 -8190.888,E2 -8190.888} C_VEL
LIN {X 0,Y 453.313,Z 650.765,A -85,B 0,C 180,E1 -8191.777,E2 -8191.777} C_VEL
LIN {X 0,Y 453.447,Z 649.81,A -85,B 0,C 180,E1 -8192.665,E2 -8192.665} C_VEL
LIN {X 0,Y 453.415,Z 648.502,A -85,B 0,C 180,E1 -8193.555,E2 -8193.555} C_VEL
LIN {X 0,Y 453.627,Z 645.693,A -85,B 0,C 180,E1 -8194.888,E2 -8194.888} C_VEL
LIN {X 0,Y 453.954,Z 641.876,A -85,B 0,C 180,E1 -8196.221,E2 -8196.221} C_VEL
LIN {X 0,Y 454.126,Z 636.801,A -85,B 0,C 180,E1 -8197.604,E2 -8197.604} C_VEL
LIN {X 0,Y 454.515,Z 630.784,A -85,B 0,C 180,E1 -8198.895,E2 -8198.895} C_VEL
LIN {X 0,Y 455.042,Z 623.009,A -85,B 0,C 180,E1 -8200.231,E2 -8200.231} C_VEL
LIN {X 0,Y 455.515,Z 613.345,A -85,B 0,C 180,E1 -8201.57,E2 -8201.57} C_VEL
LIN {X 0,Y 456.009,Z 604.316,A -85,B 0,C 180,E1 -8202.573,E2 -8202.573} C_VEL
LIN {X 0,Y 456.551,Z 593.828,A -85,B 0,C 180,E1 -8203.515,E2 -8203.515} C_VEL
LIN {X 0,Y 456.94,Z 582.332,A -85,B 0,C 180,E1 -8204.338,E2 -8204.338} C_VEL
LIN {X 0,Y 457.248,Z 571.096,A -85,B 0,C 180,E1 -8204.958,E2 -8204.958} C_VEL
LIN {X 0,Y 457.446,Z 557.931,A -85,B 0,C 180,E1 -8205.482,E2 -8205.482} C_VEL
LIN {X 0,Y 457.471,Z 544.22,A -85,B 0,C 180,E1 -8205.824,E2 -8205.824} C_VEL
LIN {X 0,Y 457.9,Z 480.226,A -85,B 0,C 180,E1 -8206.84,E2 -8206.84} C_VEL
LIN {X 0,Y 453.729,Z 468.938,A -85,B 0,C 180,E1 -8207.217,E2 -8207.217} C_VEL
LIN {X 0,Y 453.577,Z 468.143,A -85,B 0,C 180,E1 -8207.353,E2 -8207.353} C_VEL
LIN {X 0,Y 453.508,Z 467.993,A -85,B 0,C 180,E1 -8209.933,E2 -8209.933} C_VEL
LIN {X 0,Y 453.48,Z 467.984,A -85,B 0,C 180,E1 -8212.795,E2 -8212.795} C_VEL
LIN {X 0,Y 453.518,Z 467.984,A -85,B 0,C 180,E1 -8215.998,E2 -8215.998} C_VEL
LIN {X 0,Y 453.51,Z 467.982,A -85,B 0,C 180,E1 -8218.711,E2 -8218.711} C_VEL
LIN {X 0,Y 453.464,Z 467.992,A -85,B 0,C 180,E1 -8221.799,E2 -8221.799} C_VEL
LIN {X 0,Y 453.48,Z 468,A -85,B 0,C 180,E1 -8224.988,E2 -8224.988} C_VEL
LIN {X 0,Y 453.471,Z 467.993,A -85,B 0,C 180,E1 -8228.31,E2 -8228.31} C_VEL
LIN {X 0,Y 453.491,Z 467.996,A -85,B 0,C 180,E1 -8230.608,E2 -8230.608} C_VEL
LIN {X 0,Y 453.46,Z 467.991,A -85,B 0,C 180,E1 -8233.244,E2 -8233.244} C_VEL
LIN {X 0,Y 453.462,Z 467.998,A -85,B 0,C 180,E1 -8235.778,E2 -8235.778} C_VEL
LIN {X 0,Y 453.474,Z 467.99,A -85,B 0,C 180,E1 -8238.208,E2 -8238.208} C_VEL
LIN {X 0,Y 453.482,Z 467.977,A -85,B 0,C 180,E1 -8240.794,E2 -8240.794} C_VEL
LIN {X 0,Y 453.451,Z 467.998,A -85,B 0,C 180,E1 -8243.917,E2 -8243.917} C_VEL
LIN {X 0,Y 453.477,Z 467.987,A -85,B 0,C 180,E1 -8247.15,E2 -8247.15} C_VEL
LIN {X 0,Y 453.507,Z 467.971,A -85,B 0,C 180,E1 -8250.27,E2 -8250.27} C_VEL
LIN {X 0,Y 453.507,Z 467.994,A -85,B 0,C 180,E1 -8253.294,E2 -8253.294} C_VEL
LIN {X 0,Y 453.495,Z 467.989,A -85,B 0,C 180,E1 -8256.238,E2 -8256.238} C_VEL
LIN {X 0,Y 453.475,Z 467.995,A -85,B 0,C 180,E1 -8259.117,E2 -8259.117} C_VEL
LIN {X 0,Y 453.503,Z 467.989,A -85,B 0,C 180,E1 -8261.944,E2 -8261.944} C_VEL
LIN {X 0,Y 453.532,Z 467.982,A -85,B 0,C 180,E1 -8264.726,E2 -8264.726} C_VEL
LIN {X 0,Y 453.552,Z 467.983,A -85,B 0,C 180,E1 -8268.379,E2 -8268.379} C_VEL
LIN {X 0,Y 453.643,Z 467.971,A -85,B 0,C 180,E1 -8271.985,E2 -8271.985} C_VEL
LIN {X 0,Y 453.663,Z 467.97,A -85,B 0,C 180,E1 -8274.667,E2 -8274.667} C_VEL
LIN {X 0,Y 453.757,Z 467.955,A -85,B 0,C 180,E1 -8277.337,E2 -8277.337} C_VEL
LIN {X 0,Y 453.814,Z 467.952,A -85,B 0,C 180,E1 -8280,E2 -8280} C_VEL
LIN {X 0,Y 453.757,Z 467.955,A -85,B 0,C 180,E1 -8282.663,E2 -8282.663} C_VEL
LIN {X 0,Y 453.673,Z 467.968,A -85,B 0,C 180,E1 -8286.225,E2 -8286.225} C_VEL
LIN {X 0,Y 453.584,Z 467.981,A -85,B 0,C 180,E1 -8288.914,E2 -8288.914} C_VEL
LIN {X 0,Y 453.554,Z 467.982,A -85,B 0,C 180,E1 -8292.529,E2 -8292.529} C_VEL
LIN {X 0,Y 453.536,Z 467.983,A -85,B 0,C 180,E1 -8296.196,E2 -8296.196} C_VEL
LIN {X 0,Y 453.511,Z 467.975,A -85,B 0,C 180,E1 -8299.041,E2 -8299.041} C_VEL
LIN {X 0,Y 453.468,Z 468,A -85,B 0,C 180,E1 -8301.837,E2 -8301.837} C_VEL
LIN {X 0,Y 453.506,Z 467.988,A -85,B 0,C 180,E1 -8304.735,E2 -8304.735} C_VEL
LIN {X 0,Y 453.531,Z 467.987,A -85,B 0,C 180,E1 -8307.962,E2 -8307.962} C_VEL
LIN {X 0,Y 453.476,Z 467.994,A -85,B 0,C 180,E1 -8310.76,E2 -8310.76} C_VEL
LIN {X 0,Y 453.472,Z 467.995,A -85,B 0,C 180,E1 -8313.913,E2 -8313.913} C_VEL
LIN {X 0,Y 453.465,Z 467.997,A -85,B 0,C 180,E1 -8317.189,E2 -8317.189} C_VEL
LIN {X 0,Y 453.511,Z 467.991,A -85,B 0,C 180,E1 -8319.448,E2 -8319.448} C_VEL
LIN {X 0,Y 453.459,Z 467.988,A -85,B 0,C 180,E1 -8322.996,E2 -8322.996} C_VEL
LIN {X 0,Y 453.473,Z 467.993,A -85,B 0,C 180,E1 -8325.781,E2 -8325.781} C_VEL
LIN {X 0,Y 453.493,Z 467.99,A -85,B 0,C 180,E1 -8328.212,E2 -8328.212} C_VEL
LIN {X 0,Y 453.523,Z 467.988,A -85,B 0,C 180,E1 -8330.789,E2 -8330.789} C_VEL
LIN {X 0,Y 453.454,Z 467.994,A -85,B 0,C 180,E1 -8333.918,E2 -8333.918} C_VEL
LIN {X 0,Y 453.482,Z 467.993,A -85,B 0,C 180,E1 -8337.152,E2 -8337.152} C_VEL
LIN {X 0,Y 453.523,Z 468.147,A -85,B 0,C 180,E1 -8339.122,E2 -8339.122} C_VEL
LIN {X 0,Y 456.631,Z 481.873,A -85,B 0,C 180,E1 -8341.317,E2 -8341.317} C_VEL
LIN {X 0,Y 457.615,Z 486.814,A -85,B 0,C 180,E1 -8342.069,E2 -8342.069} C_VEL
LIN {X 0,Y 456.665,Z 507.831,A -85,B 0,C 180,E1 -8344.98,E2 -8344.98} C_VEL
LIN {X 0,Y 455.618,Z 530.834,A -85,B 0,C 180,E1 -8348.117,E2 -8348.117} C_VEL
LIN {X 0,Y 454.685,Z 554.152,A -85,B 0,C 180,E1 -8351.293,E2 -8351.293} C_VEL
LIN {X 0,Y 454.435,Z 562.446,A -85,B 0,C 180,E1 -8352.401,E2 -8352.401} C_VEL
LIN {X 0,Y 457.385,Z 589.793,A -85,B 0,C 180,E1 -8352.968,E2 -8352.968} C_VEL
LIN {X 0,Y 456.689,Z 672.857,A -85,B 0,C 180,E1 -8354.291,E2 -8354.291} C_VEL
LIN {X 0,Y 456.224,Z 686.185,A -85,B 0,C 180,E1 -8354.676,E2 -8354.676} C_VEL
LIN {X 0,Y 455.673,Z 698.426,A -85,B 0,C 180,E1 -8355.2,E2 -8355.2} C_VEL
LIN {X 0,Y 455.063,Z 710.82,A -85,B 0,C 180,E1 -8355.922,E2 -8355.922} C_VEL
LIN {X 0,Y 454.484,Z 721.786,A -85,B 0,C 180,E1 -8356.749,E2 -8356.749} C_VEL
LIN {X 0,Y 454.04,Z 733.176,A -85,B 0,C 180,E1 -8357.825,E2 -8357.825} C_VEL
LIN {X 0,Y 453.561,Z 741.86,A -85,B 0,C 180,E1 -8358.832,E2 -8358.832} C_VEL
LIN {X 0,Y 453.209,Z 749.904,A -85,B 0,C 180,E1 -8359.953,E2 -8359.953} C_VEL
LIN {X 0,Y 452.962,Z 757.791,A -85,B 0,C 180,E1 -8361.299,E2 -8361.299} C_VEL
LIN {X 0,Y 452.859,Z 765.085,A -85,B 0,C 180,E1 -8362.868,E2 -8362.868} C_VEL
LIN {X 0,Y 452.838,Z 769.952,A -85,B 0,C 180,E1 -8364.21,E2 -8364.21} C_VEL
LIN {X 0,Y 452.858,Z 773.679,A -85,B 0,C 180,E1 -8365.55,E2 -8365.55} C_VEL
LIN {X 0,Y 452.877,Z 775.604,A -85,B 0,C 180,E1 -8366.441,E2 -8366.441} C_VEL
LIN {X 0,Y 452.872,Z 777.046,A -85,B 0,C 180,E1 -8367.332,E2 -8367.332} C_VEL
LIN {X 0,Y 453.023,Z 778.724,A -85,B 0,C 180,E1 -8369.111,E2 -8369.111} C_VEL
LIN {X 0,Y 453.025,Z 778.947,A -85,B 0,C 180,E1 -8370,E2 -8370} C_VEL
LIN {X 0,Y 453.023,Z 778.724,A -85,B 0,C 180,E1 -8370.889,E2 -8370.889} C_VEL
LIN {X 0,Y 452.872,Z 777.049,A -85,B 0,C 180,E1 -8372.668,E2 -8372.668} C_VEL
LIN {X 0,Y 452.877,Z 775.607,A -85,B 0,C 180,E1 -8373.559,E2 -8373.559} C_VEL
LIN {X 0,Y 452.854,Z 772.575,A -85,B 0,C 180,E1 -8374.896,E2 -8374.896} C_VEL
LIN {X 0,Y 452.83,Z 768.473,A -85,B 0,C 180,E1 -8376.237,E2 -8376.237} C_VEL
LIN {X 0,Y 452.886,Z 762.181,A -85,B 0,C 180,E1 -8377.804,E2 -8377.804} C_VEL
LIN {X 0,Y 453.033,Z 755.328,A -85,B 0,C 180,E1 -8379.149,E2 -8379.149} C_VEL
LIN {X 0,Y 453.327,Z 746.857,A -85,B 0,C 180,E1 -8380.495,E2 -8380.495} C_VEL
LIN {X 0,Y 453.666,Z 738.191,A -85,B 0,C 180,E1 -8381.618,E2 -8381.618} C_VEL
LIN {X 0,Y 454.243,Z 728.499,A -85,B 0,C 180,E1 -8382.646,E2 -8382.646} C_VEL
LIN {X 0,Y 454.772,Z 717.02,A -85,B 0,C 180,E1 -8383.631,E2 -8383.631} C_VEL
LIN {X 0,Y 455.354,Z 705.523,A -85,B 0,C 180,E1 -8384.411,E2 -8384.411} C_VEL
LIN {X 0,Y 455.892,Z 693.749,A -85,B 0,C 180,E1 -8385.021,E2 -8385.021} C_VEL
LIN {X 0,Y 456.479,Z 680.237,A -85,B 0,C 180,E1 -8385.516,E2 -8385.516} C_VEL
LIN {X 0,Y 456.793,Z 666.892,A -85,B 0,C 180,E1 -8385.819,E2 -8385.819} C_VEL
LIN {X 0,Y 457.301,Z 588.744,A -85,B 0,C 180,E1 -8387.05,E2 -8387.05} C_VEL
LIN {X 0,Y 454.398,Z 562.448,A -85,B 0,C 180,E1 -8387.598,E2 -8387.598} C_VEL
LIN {X 0,Y 455.296,Z 538.796,A -85,B 0,C 180,E1 -8390.795,E2 -8390.795} C_VEL
LIN {X 0,Y 456.331,Z 514.633,A -85,B 0,C 180,E1 -8394.087,E2 -8394.087} C_VEL
LIN {X 0,Y 457.548,Z 490.266,A -85,B 0,C 180,E1 -8397.438,E2 -8397.438} C_VEL
LIN {X 0,Y 457.597,Z 486.771,A -85,B 0,C 180,E1 -8397.932,E2 -8397.932} C_VEL
LIN {X 0,Y 455.024,Z 474.327,A -85,B 0,C 180,E1 -8399.853,E2 -8399.853} C_VEL
LIN {X 0,Y 453.522,Z 468.13,A -85,B 0,C 180,E1 -8400.878,E2 -8400.878} C_VEL
LIN {X 0,Y 453.475,Z 467.994,A -85,B 0,C 180,E1 -8403.912,E2 -8403.912} C_VEL
LIN {X 0,Y 453.467,Z 467.994,A -85,B 0,C 180,E1 -8407.187,E2 -8407.187} C_VEL
LIN {X 0,Y 453.526,Z 467.988,A -85,B 0,C 180,E1 -8409.445,E2 -8409.445} C_VEL
LIN {X 0,Y 453.488,Z 467.995,A -85,B 0,C 180,E1 -8412.991,E2 -8412.991} C_VEL
LIN {X 0,Y 453.461,Z 467.982,A -85,B 0,C 180,E1 -8415.778,E2 -8415.778} C_VEL
LIN {X 0,Y 453.474,Z 467.994,A -85,B 0,C 180,E1 -8418.209,E2 -8418.209} C_VEL
LIN {X 0,Y 453.51,Z 467.988,A -85,B 0,C 180,E1 -8420.789,E2 -8420.789} C_VEL
LIN {X 0,Y 453.451,Z 468,A -85,B 0,C 180,E1 -8423.917,E2 -8423.917} C_VEL
LIN {X 0,Y 453.476,Z 467.988,A -85,B 0,C 180,E1 -8427.151,E2 -8427.151} C_VEL
LIN {X 0,Y 453.507,Z 467.998,A -85,B 0,C 180,E1 -8430.271,E2 -8430.271} C_VEL
LIN {X 0,Y 453.506,Z 467.979,A -85,B 0,C 180,E1 -8433.294,E2 -8433.294} C_VEL
LIN {X 0,Y 453.495,Z 467.996,A -85,B 0,C 180,E1 -8436.238,E2 -8436.238} C_VEL
LIN {X 0,Y 453.474,Z 467.988,A -85,B 0,C 180,E1 -8439.117,E2 -8439.117} C_VEL
LIN {X 0,Y 453.502,Z 467.977,A -85,B 0,C 180,E1 -8441.944,E2 -8441.944} C_VEL
LIN {X 0,Y 453.53,Z 467.992,A -85,B 0,C 180,E1 -8444.726,E2 -8444.726} C_VEL
LIN {X 0,Y 453.552,Z 467.984,A -85,B 0,C 180,E1 -8448.379,E2 -8448.379} C_VEL
LIN {X 0,Y 453.642,Z 467.975,A -85,B 0,C 180,E1 -8451.985,E2 -8451.985} C_VEL
LIN {X 0,Y 453.669,Z 467.967,A -85,B 0,C 180,E1 -8454.667,E2 -8454.667} C_VEL
LIN {X 0,Y 453.757,Z 467.957,A -85,B 0,C 180,E1 -8457.337,E2 -8457.337} C_VEL
LIN {X 0,Y 453.814,Z 467.953,A -85,B 0,C 180,E1 -8460,E2 -8460} C_VEL
LIN {X 0,Y 453.757,Z 467.956,A -85,B 0,C 180,E1 -8462.663,E2 -8462.663} C_VEL
LIN {X 0,Y 453.675,Z 467.971,A -85,B 0,C 180,E1 -8466.225,E2 -8466.225} C_VEL
LIN {X 0,Y 453.584,Z 467.976,A -85,B 0,C 180,E1 -8468.914,E2 -8468.914} C_VEL
LIN {X 0,Y 453.554,Z 467.989,A -85,B 0,C 180,E1 -8472.529,E2 -8472.529} C_VEL
LIN {X 0,Y 453.536,Z 467.981,A -85,B 0,C 180,E1 -8476.196,E2 -8476.196} C_VEL
LIN {X 0,Y 453.512,Z 467.994,A -85,B 0,C 180,E1 -8479.041,E2 -8479.041} C_VEL
LIN {X 0,Y 453.468,Z 467.99,A -85,B 0,C 180,E1 -8481.837,E2 -8481.837} C_VEL
LIN {X 0,Y 453.507,Z 467.996,A -85,B 0,C 180,E1 -8484.735,E2 -8484.735} C_VEL
LIN {X 0,Y 453.532,Z 467.981,A -85,B 0,C 180,E1 -8487.962,E2 -8487.962} C_VEL
LIN {X 0,Y 453.476,Z 467.973,A -85,B 0,C 180,E1 -8490.76,E2 -8490.76} C_VEL
LIN {X 0,Y 453.472,Z 467.991,A -85,B 0,C 180,E1 -8493.913,E2 -8493.913} C_VEL
LIN {X 0,Y 453.465,Z 467.995,A -85,B 0,C 180,E1 -8497.189,E2 -8497.189} C_VEL
LIN {X 0,Y 453.489,Z 467.976,A -85,B 0,C 180,E1 -8500.61,E2 -8500.61} C_VEL
LIN {X 0,Y 453.452,Z 468.002,A -85,B 0,C 180,E1 -8503.245,E2 -8503.245} C_VEL
LIN {X 0,Y 453.469,Z 467.991,A -85,B 0,C 180,E1 -8505.781,E2 -8505.781} C_VEL
LIN {X 0,Y 453.478,Z 467.985,A -85,B 0,C 180,E1 -8508.21,E2 -8508.21} C_VEL
LIN {X 0,Y 453.516,Z 467.995,A -85,B 0,C 180,E1 -8510.79,E2 -8510.79} C_VEL
LIN {X 0,Y 453.454,Z 467.978,A -85,B 0,C 180,E1 -8513.918,E2 -8513.918} C_VEL
LIN {X 0,Y 453.482,Z 467.977,A -85,B 0,C 180,E1 -8517.152,E2 -8517.152} C_VEL
LIN {X 0,Y 453.475,Z 467.997,A -85,B 0,C 180,E1 -8520.269,E2 -8520.269} C_VEL
LIN {X 0,Y 453.506,Z 467.975,A -85,B 0,C 180,E1 -8523.295,E2 -8523.295} C_VEL
LIN {X 0,Y 453.504,Z 467.992,A -85,B 0,C 180,E1 -8526.239,E2 -8526.239} C_VEL
LIN {X 0,Y 453.485,Z 467.994,A -85,B 0,C 180,E1 -8529.118,E2 -8529.118} C_VEL
LIN {X 0,Y 453.529,Z 467.941,A -85,B 0,C 180,E1 -8532.412,E2 -8532.412} C_VEL
LIN {X 0,Y 453.586,Z 468.305,A -85,B 0,C 180,E1 -8532.792,E2 -8532.792} C_VEL
LIN {X 0,Y 453.958,Z 469.626,A -85,B 0,C 180,E1 -8532.916,E2 -8532.916} C_VEL
LIN {X 0,Y 457.905,Z 480.124,A -85,B 0,C 180,E1 -8533.253,E2 -8533.253} C_VEL
LIN {X 0,Y 457.513,Z 548.271,A -85,B 0,C 180,E1 -8534.349,E2 -8534.349} C_VEL
LIN {X 0,Y 457.51,Z 549.705,A -85,B 0,C 180,E1 -8534.383,E2 -8534.383} C_VEL
LIN {X 0,Y 456.39,Z 557.375,A -85,B 0,C 180,E1 -8534.553,E2 -8534.553} C_VEL
LIN {X 0,Y 452.691,Z 568.49,A -85,B 0,C 180,E1 -8534.828,E2 -8534.828} C_VEL
LIN {X 0,Y 450.671,Z 575.828,A -85,B 0,C 180,E1 -8535.11,E2 -8535.11} C_VEL
LIN {X 0,Y 450.251,Z 579.404,A -85,B 0,C 180,E1 -8535.298,E2 -8535.298} C_VEL
LIN {X 0,Y 449.906,Z 591.439,A -85,B 0,C 180,E1 -8536.102,E2 -8536.102} C_VEL
LIN {X 0,Y 449.327,Z 600.872,A -85,B 0,C 180,E1 -8536.892,E2 -8536.892} C_VEL
LIN {X 0,Y 448.881,Z 609.718,A -85,B 0,C 180,E1 -8537.798,E2 -8537.798} C_VEL
LIN {X 0,Y 448.385,Z 618.777,A -85,B 0,C 180,E1 -8538.93,E2 -8538.93} C_VEL
LIN {X 0,Y 447.867,Z 627.549,A -85,B 0,C 180,E1 -8540.289,E2 -8540.289} C_VEL
LIN {X 0,Y 447.454,Z 633.735,A -85,B 0,C 180,E1 -8541.464,E2 -8541.464} C_VEL
LIN {X 0,Y 447.146,Z 639.351,A -85,B 0,C 180,E1 -8542.777,E2 -8542.777} C_VEL
LIN {X 0,Y 446.778,Z 643.974,A -85,B 0,C 180,E1 -8544.132,E2 -8544.132} C_VEL
LIN {X 0,Y 446.535,Z 647.505,A -85,B 0,C 180,E1 -8545.487,E2 -8545.487} C_VEL
LIN {X 0,Y 446.404,Z 649.33,A -85,B 0,C 180,E1 -8546.39,E2 -8546.39} C_VEL
LIN {X 0,Y 446.431,Z 650.688,A -85,B 0,C 180,E1 -8547.293,E2 -8547.293} C_VEL
LIN {X 0,Y 446.291,Z 651.674,A -85,B 0,C 180,E1 -8548.195,E2 -8548.195} C_VEL
LIN {X 0,Y 446.37,Z 652.259,A -85,B 0,C 180,E1 -8549.098,E2 -8549.098} C_VEL
LIN {X 0,Y 446.354,Z 652.49,A -85,B 0,C 180,E1 -8550,E2 -8550} C_VEL
LIN {X 0,Y 446.37,Z 652.307,A -85,B 0,C 180,E1 -8550.902,E2 -8550.902} C_VEL
LIN {X 0,Y 446.291,Z 651.752,A -85,B 0,C 180,E1 -8551.805,E2 -8551.805} C_VEL
LIN {X 0,Y 446.43,Z 650.797,A -85,B 0,C 180,E1 -8552.707,E2 -8552.707} C_VEL
LIN {X 0,Y 446.398,Z 649.49,A -85,B 0,C 180,E1 -8553.611,E2 -8553.611} C_VEL
LIN {X 0,Y 446.622,Z 646.681,A -85,B 0,C 180,E1 -8554.965,E2 -8554.965} C_VEL
LIN {X 0,Y 446.97,Z 642.862,A -85,B 0,C 180,E1 -8556.319,E2 -8556.319} C_VEL
LIN {X 0,Y 447.161,Z 637.788,A -85,B 0,C 180,E1 -8557.723,E2 -8557.723} C_VEL
LIN {X 0,Y 447.575,Z 631.77,A -85,B 0,C 180,E1 -8559.034,E2 -8559.034} C_VEL
LIN {X 0,Y 448.128,Z 623.995,A -85,B 0,C 180,E1 -8560.39,E2 -8560.39} C_VEL
LIN {X 0,Y 448.63,Z 614.33,A -85,B 0,C 180,E1 -8561.75,E2 -8561.75} C_VEL
LIN {X 0,Y 449.15,Z 605.3,A -85,B 0,C 180,E1 -8562.769,E2 -8562.769} C_VEL
LIN {X 0,Y 449.72,Z 594.811,A -85,B 0,C 180,E1 -8563.724,E2 -8563.724} C_VEL
LIN {X 0,Y 450.124,Z 583.161,A -85,B 0,C 180,E1 -8564.57,E2 -8564.57} C_VEL
LIN {X 0,Y 450.48,Z 571.741,A -85,B 0,C 180,E1 -8565.206,E2 -8565.206} C_VEL
LIN {X 0,Y 450.659,Z 558.908,A -85,B 0,C 180,E1 -8565.721,E2 -8565.721} C_VEL
LIN {X 0,Y 450.69,Z 545.189,A -85,B 0,C 180,E1 -8566.068,E2 -8566.068} C_VEL
LIN {X 0,Y 451.156,Z 481.764,A -85,B 0,C 180,E1 -8567.09,E2 -8567.09} C_VEL
LIN {X 0,Y 446.724,Z 469.919,A -85,B 0,C 180,E1 -8567.49,E2 -8567.49} C_VEL
LIN {X 0,Y 446.506,Z 468.959,A -85,B 0,C 180,E1 -8567.667,E2 -8567.667} C_VEL
LIN {X 0,Y 446.447,Z 468.874,A -85,B 0,C 180,E1 -8570.262,E2 -8570.262} C_VEL
LIN {X 0,Y 446.43,Z 468.866,A -85,B 0,C 180,E1 -8573.176,E2 -8573.176} C_VEL
LIN {X 0,Y 446.476,Z 468.857,A -85,B 0,C 180,E1 -8576.202,E2 -8576.202} C_VEL
LIN {X 0,Y 446.449,Z 468.869,A -85,B 0,C 180,E1 -8579.209,E2 -8579.209} C_VEL
LIN {X 0,Y 446.422,Z 468.87,A -85,B 0,C 180,E1 -8582.361,E2 -8582.361} C_VEL
LIN {X 0,Y 446.419,Z 468.871,A -85,B 0,C 180,E1 -8585.625,E2 -8585.625} C_VEL
LIN {X 0,Y 446.455,Z 468.874,A -85,B 0,C 180,E1 -8589.025,E2 -8589.025} C_VEL
LIN {X 0,Y 446.433,Z 468.863,A -85,B 0,C 180,E1 -8592.277,E2 -8592.277} C_VEL
LIN {X 0,Y 446.451,Z 468.874,A -85,B 0,C 180,E1 -8595.102,E2 -8595.102} C_VEL
LIN {X 0,Y 446.423,Z 468.87,A -85,B 0,C 180,E1 -8598.608,E2 -8598.608} C_VEL
LIN {X 0,Y 446.434,Z 468.856,A -85,B 0,C 180,E1 -8600.972,E2 -8600.972} C_VEL
LIN {X 0,Y 446.416,Z 468.874,A -85,B 0,C 180,E1 -8604.373,E2 -8604.373} C_VEL
LIN {X 0,Y 446.416,Z 468.859,A -85,B 0,C 180,E1 -8607.638,E2 -8607.638} C_VEL
LIN {X 0,Y 446.463,Z 468.85,A -85,B 0,C 180,E1 -8610.791,E2 -8610.791} C_VEL
LIN {X 0,Y 446.47,Z 468.868,A -85,B 0,C 180,E1 -8613.848,E2 -8613.848} C_VEL
LIN {X 0,Y 446.421,Z 468.873,A -85,B 0,C 180,E1 -8616.823,E2 -8616.823} C_VEL
LIN {X 0,Y 446.436,Z 468.873,A -85,B 0,C 180,E1 -8619.737,E2 -8619.737} C_VEL
LIN {X 0,Y 446.455,Z 468.867,A -85,B 0,C 180,E1 -8622.597,E2 -8622.597} C_VEL
LIN {X 0,Y 446.463,Z 468.87,A -85,B 0,C 180,E1 -8625.412,E2 -8625.412} C_VEL
LIN {X 0,Y 446.51,Z 468.861,A -85,B 0,C 180,E1 -8628.193,E2 -8628.193} C_VEL
LIN {X 0,Y 446.591,Z 468.851,A -85,B 0,C 180,E1 -8631.858,E2 -8631.858} C_VEL
LIN {X 0,Y 446.637,Z 468.845,A -85,B 0,C 180,E1 -8634.582,E2 -8634.582} C_VEL
LIN {X 0,Y 446.701,Z 468.833,A -85,B 0,C 180,E1 -8637.295,E2 -8637.295} C_VEL
LIN {X 0,Y 446.785,Z 468.827,A -85,B 0,C 180,E1 -8640,E2 -8640} C_VEL
LIN {X 0,Y 446.701,Z 468.834,A -85,B 0,C 180,E1 -8642.705,E2 -8642.705} C_VEL
LIN {X 0,Y 446.642,Z 468.844,A -85,B 0,C 180,E1 -8646.324,E2 -8646.324} C_VEL
LIN {X 0,Y 446.529,Z 468.861,A -85,B 0,C 180,E1 -8649.056,E2 -8649.056} C_VEL
LIN {X 0,Y 446.512,Z 468.859,A -85,B 0,C 180,E1 -8652.73,E2 -8652.73} C_VEL
LIN {X 0,Y 446.487,Z 468.861,A -85,B 0,C 180,E1 -8656.228,E2 -8656.228} C_VEL
LIN {X 0,Y 446.461,Z 468.854,A -85,B 0,C 180,E1 -8659.304,E2 -8659.304} C_VEL
LIN {X 0,Y 446.409,Z 468.876,A -85,B 0,C 180,E1 -8662.2,E2 -8662.2} C_VEL
LIN {X 0,Y 446.451,Z 468.87,A -85,B 0,C 180,E1 -8665.153,E2 -8665.153} C_VEL
LIN {X 0,Y 446.477,Z 468.865,A -85,B 0,C 180,E1 -8668.179,E2 -8668.179} C_VEL
LIN {X 0,Y 446.424,Z 468.876,A -85,B 0,C 180,E1 -8671.3,E2 -8671.3} C_VEL
LIN {X 0,Y 446.424,Z 468.871,A -85,B 0,C 180,E1 -8674.524,E2 -8674.524} C_VEL
LIN {X 0,Y 446.425,Z 468.871,A -85,B 0,C 180,E1 -8678.083,E2 -8678.083} C_VEL
LIN {X 0,Y 446.422,Z 468.874,A -85,B 0,C 180,E1 -8680.918,E2 -8680.918} C_VEL
LIN {X 0,Y 446.397,Z 468.861,A -85,B 0,C 180,E1 -8683.847,E2 -8683.847} C_VEL
LIN {X 0,Y 446.443,Z 468.874,A -85,B 0,C 180,E1 -8686.398,E2 -8686.398} C_VEL
LIN {X 0,Y 446.465,Z 468.86,A -85,B 0,C 180,E1 -8689.806,E2 -8689.806} C_VEL
LIN {X 0,Y 446.429,Z 468.875,A -85,B 0,C 180,E1 -8692.124,E2 -8692.124} C_VEL
LIN {X 0,Y 446.429,Z 468.879,A -85,B 0,C 180,E1 -8695.478,E2 -8695.478} C_VEL
LIN {X 0,Y 446.491,Z 469.074,A -85,B 0,C 180,E1 -8698.87,E2 -8698.87} C_VEL
LIN {X 0,Y 449.854,Z 483.9,A -85,B 0,C 180,E1 -8701.269,E2 -8701.269} C_VEL
LIN {X 0,Y 450.739,Z 489.421,A -85,B 0,C 180,E1 -8702.111,E2 -8702.111} C_VEL
LIN {X 0,Y 449.581,Z 511.995,A -85,B 0,C 180,E1 -8705.282,E2 -8705.282} C_VEL
LIN {X 0,Y 448.489,Z 534.429,A -85,B 0,C 180,E1 -8708.393,E2 -8708.393} C_VEL
LIN {X 0,Y 447.6,Z 556.53,A -85,B 0,C 180,E1 -8711.461,E2 -8711.461} C_VEL
LIN {X 0,Y 447.446,Z 561.511,A -85,B 0,C 180,E1 -8712.121,E2 -8712.121} C_VEL
LIN {X 0,Y 450.567,Z 590.704,A -85,B 0,C 180,E1 -8712.734,E2 -8712.734} C_VEL
LIN {X 0,Y 449.816,Z 671.863,A -85,B 0,C 180,E1 -8714.045,E2 -8714.045} C_VEL
LIN {X 0,Y 449.382,Z 685.194,A -85,B 0,C 180,E1 -8714.437,E2 -8714.437} C_VEL
LIN {X 0,Y 448.775,Z 697.428,A -85,B 0,C 180,E1 -8714.967,E2 -8714.967} C_VEL
LIN {X 0,Y 448.148,Z 709.821,A -85,B 0,C 180,E1 -8715.701,E2 -8715.701} C_VEL
LIN {X 0,Y 447.49,Z 721.301,A -85,B 0,C 180,E1 -8716.584,E2 -8716.584} C_VEL
LIN {X 0,Y 447.061,Z 732.174,A -85,B 0,C 180,E1 -8717.632,E2 -8717.632} C_VEL
LIN {X 0,Y 446.527,Z 740.854,A -85,B 0,C 180,E1 -8718.654,E2 -8718.654} C_VEL
LIN {X 0,Y 446.164,Z 748.899,A -85,B 0,C 180,E1 -8719.793,E2 -8719.793} C_VEL
LIN {X 0,Y 445.878,Z 756.784,A -85,B 0,C 180,E1 -8721.16,E2 -8721.16} C_VEL
LIN {X 0,Y 445.812,Z 762.209,A -85,B 0,C 180,E1 -8722.299,E2 -8722.299} C_VEL
LIN {X 0,Y 445.761,Z 767.476,A -85,B 0,C 180,E1 -8723.664,E2 -8723.664} C_VEL
LIN {X 0,Y 445.805,Z 771.58,A -85,B 0,C 180,E1 -8725.026,E2 -8725.026} C_VEL
LIN {X 0,Y 445.835,Z 774.612,A -85,B 0,C 180,E1 -8726.385,E2 -8726.385} C_VEL
LIN {X 0,Y 445.827,Z 776.054,A -85,B 0,C 180,E1 -8727.289,E2 -8727.289} C_VEL
LIN {X 0,Y 446.002,Z 777.737,A -85,B 0,C 180,E1 -8729.097,E2 -8729.097} C_VEL
LIN {X 0,Y 446.006,Z 777.96,A -85,B 0,C 180,E1 -8730,E2 -8730} C_VEL
LIN {X 0,Y 446.002,Z 777.737,A -85,B 0,C 180,E1 -8730.903,E2 -8730.903} C_VEL
LIN {X 0,Y 445.827,Z 776.057,A -85,B 0,C 180,E1 -8732.711,E2 -8732.711} C_VEL
LIN {X 0,Y 445.835,Z 774.615,A -85,B 0,C 180,E1 -8733.615,E2 -8733.615} C_VEL
LIN {X 0,Y 445.805,Z 771.58,A -85,B 0,C 180,E1 -8734.974,E2 -8734.974} C_VEL
LIN {X 0,Y 445.75,Z 766.402,A -85,B 0,C 180,E1 -8736.634,E2 -8736.634} C_VEL
LIN {X 0,Y 445.849,Z 760.139,A -85,B 0,C 180,E1 -8738.156,E2 -8738.156} C_VEL
LIN {X 0,Y 446.021,Z 753.056,A -85,B 0,C 180,E1 -8739.523,E2 -8739.523} C_VEL
LIN {X 0,Y 446.36,Z 744.224,A -85,B 0,C 180,E1 -8740.891,E2 -8740.891} C_VEL
LIN {X 0,Y 446.815,Z 735.207,A -85,B 0,C 180,E1 -8742.029,E2 -8742.029} C_VEL
LIN {X 0,Y 447.353,Z 724.343,A -85,B 0,C 180,E1 -8743.147,E2 -8743.147} C_VEL
LIN {X 0,Y 447.944,Z 712.995,A -85,B 0,C 180,E1 -8744.074,E2 -8744.074} C_VEL
LIN {X 0,Y 448.672,Z 700.565,A -85,B 0,C 180,E1 -8744.862,E2 -8744.862} C_VEL
LIN {X 0,Y 449.227,Z 688.821,A -85,B 0,C 180,E1 -8745.424,E2 -8745.424} C_VEL
LIN {X 0,Y 449.733,Z 676.358,A -85,B 0,C 180,E1 -8745.842,E2 -8745.842} C_VEL
LIN {X 0,Y 450.009,Z 660.5,A -85,B 0,C 180,E1 -8746.152,E2 -8746.152} C_VEL
LIN {X 0,Y 450.422,Z 588.994,A -85,B 0,C 180,E1 -8747.297,E2 -8747.297} C_VEL
LIN {X 0,Y 447.425,Z 561.448,A -85,B 0,C 180,E1 -8747.88,E2 -8747.88} C_VEL
LIN {X 0,Y 448.336,Z 537.821,A -85,B 0,C 180,E1 -8751.133,E2 -8751.133} C_VEL
LIN {X 0,Y 449.481,Z 513.7,A -85,B 0,C 180,E1 -8754.478,E2 -8754.478} C_VEL
LIN {X 0,Y 450.743,Z 489.367,A -85,B 0,C 180,E1 -8757.888,E2 -8757.888} C_VEL
LIN {X 0,Y 449.191,Z 480.414,A -85,B 0,C 180,E1 -8759.27,E2 -8759.27} C_VEL
LIN {X 0,Y 446.483,Z 468.983,A -85,B 0,C 180,E1 -8761.162,E2 -8761.162} C_VEL
LIN {X 0,Y 446.427,Z 468.88,A -85,B 0,C 180,E1 -8764.522,E2 -8764.522} C_VEL
LIN {X 0,Y 446.432,Z 468.877,A -85,B 0,C 180,E1 -8768.082,E2 -8768.082} C_VEL
LIN {X 0,Y 446.444,Z 468.866,A -85,B 0,C 180,E1 -8770.92,E2 -8770.92} C_VEL
LIN {X 0,Y 446.441,Z 468.876,A -85,B 0,C 180,E1 -8773.84,E2 -8773.84} C_VEL
LIN {X 0,Y 446.395,Z 468.862,A -85,B 0,C 180,E1 -8776.403,E2 -8776.403} C_VEL
LIN {X 0,Y 446.422,Z 468.874,A -85,B 0,C 180,E1 -8779.082,E2 -8779.082} C_VEL
LIN {X 0,Y 446.425,Z 468.87,A -85,B 0,C 180,E1 -8781.918,E2 -8781.918} C_VEL
LIN {X 0,Y 446.424,Z 468.871,A -85,B 0,C 180,E1 -8785.476,E2 -8785.476} C_VEL
LIN {X 0,Y 446.424,Z 468.877,A -85,B 0,C 180,E1 -8788.7,E2 -8788.7} C_VEL
LIN {X 0,Y 446.477,Z 468.865,A -85,B 0,C 180,E1 -8791.821,E2 -8791.821} C_VEL
LIN {X 0,Y 446.451,Z 468.87,A -85,B 0,C 180,E1 -8794.847,E2 -8794.847} C_VEL
LIN {X 0,Y 446.44,Z 468.875,A -85,B 0,C 180,E1 -8798.245,E2 -8798.245} C_VEL
LIN {X 0,Y 446.448,Z 468.854,A -85,B 0,C 180,E1 -8801.649,E2 -8801.649} C_VEL
LIN {X 0,Y 446.498,Z 468.868,A -85,B 0,C 180,E1 -8804.479,E2 -8804.479} C_VEL
LIN {X 0,Y 446.509,Z 468.862,A -85,B 0,C 180,E1 -8808.193,E2 -8808.193} C_VEL
LIN {X 0,Y 446.591,Z 468.852,A -85,B 0,C 180,E1 -8811.858,E2 -8811.858} C_VEL
LIN {X 0,Y 446.643,Z 468.843,A -85,B 0,C 180,E1 -8814.583,E2 -8814.583} C_VEL
LIN {X 0,Y 446.701,Z 468.836,A -85,B 0,C 180,E1 -8817.295,E2 -8817.295} C_VEL
LIN {X 0,Y 446.785,Z 468.829,A -85,B 0,C 180,E1 -8820,E2 -8820} C_VEL
LIN {X 0,Y 446.701,Z 468.834,A -85,B 0,C 180,E1 -8822.705,E2 -8822.705} C_VEL
LIN {X 0,Y 446.643,Z 468.848,A -85,B 0,C 180,E1 -8826.324,E2 -8826.324} C_VEL
LIN {X 0,Y 446.53,Z 468.853,A -85,B 0,C 180,E1 -8829.056,E2 -8829.056} C_VEL
LIN {X 0,Y 446.512,Z 468.869,A -85,B 0,C 180,E1 -8832.73,E2 -8832.73} C_VEL
LIN {X 0,Y 446.487,Z 468.859,A -85,B 0,C 180,E1 -8836.228,E2 -8836.228} C_VEL
LIN {X 0,Y 446.461,Z 468.87,A -85,B 0,C 180,E1 -8839.304,E2 -8839.304} C_VEL
LIN {X 0,Y 446.41,Z 468.87,A -85,B 0,C 180,E1 -8842.2,E2 -8842.2} C_VEL
LIN {X 0,Y 446.451,Z 468.873,A -85,B 0,C 180,E1 -8845.153,E2 -8845.153} C_VEL
LIN {X 0,Y 446.477,Z 468.861,A -85,B 0,C 180,E1 -8848.179,E2 -8848.179} C_VEL
LIN {X 0,Y 446.413,Z 468.855,A -85,B 0,C 180,E1 -8851.301,E2 -8851.301} C_VEL
LIN {X 0,Y 446.424,Z 468.872,A -85,B 0,C 180,E1 -8854.524,E2 -8854.524} C_VEL
LIN {X 0,Y 446.423,Z 468.868,A -85,B 0,C 180,E1 -8858.082,E2 -8858.082} C_VEL
LIN {X 0,Y 446.422,Z 468.86,A -85,B 0,C 180,E1 -8860.918,E2 -8860.918} C_VEL
LIN {X 0,Y 446.398,Z 468.876,A -85,B 0,C 180,E1 -8863.847,E2 -8863.847} C_VEL
LIN {X 0,Y 446.417,Z 468.87,A -85,B 0,C 180,E1 -8866.401,E2 -8866.401} C_VEL
LIN {X 0,Y 446.449,Z 468.87,A -85,B 0,C 180,E1 -8869.804,E2 -8869.804} C_VEL
LIN {X 0,Y 446.427,Z 468.869,A -85,B 0,C 180,E1 -8872.124,E2 -8872.124} C_VEL
LIN {X 0,Y 446.428,Z 468.838,A -85,B 0,C 180,E1 -8875.478,E2 -8875.478} C_VEL
LIN {X 0,Y 446.416,Z 468.874,A -85,B 0,C 180,E1 -8878.701,E2 -8878.701} C_VEL
LIN {X 0,Y 446.485,Z 468.854,A -85,B 0,C 180,E1 -8881.822,E2 -8881.822} C_VEL
LIN {X 0,Y 446.458,Z 468.868,A -85,B 0,C 180,E1 -8884.848,E2 -8884.848} C_VEL
LIN {X 0,Y 446.449,Z 468.859,A -85,B 0,C 180,E1 -8888.246,E2 -8888.246} C_VEL
LIN {X 0,Y 446.458,Z 468.831,A -85,B 0,C 180,E1 -8891.65,E2 -8891.65} C_VEL
LIN {X 0,Y 446.545,Z 469.085,A -85,B 0,C 180,E1 -8892.483,E2 -8892.483} C_VEL
LIN {X 0,Y 446.815,Z 470.226,A -85,B 0,C 180,E1 -8892.623,E2 -8892.623} C_VEL
LIN {X 0,Y 451.122,Z 481.655,A -85,B 0,C 180,E1 -8893.001,E2 -8893.001} C_VEL
LIN {X 0,Y 450.74,Z 550.186,A -85,B 0,C 180,E1 -8894.129,E2 -8894.129} C_VEL
LIN {X 0,Y 450.651,Z 562.764,A -85,B 0,C 180,E1 -8894.511,E2 -8894.511} C_VEL
LIN {X 0,Y 450.365,Z 574.39,A -85,B 0,C 180,E1 -8895.022,E2 -8895.022} C_VEL
LIN {X 0,Y 450.251,Z 579.404,A -85,B 0,C 180,E1 -8895.298,E2 -8895.298} C_VEL
LIN {X 0,Y 449.444,Z 584.778,A -85,B 0,C 180,E1 -8895.601,E2 -8895.601} C_VEL
LIN {X 0,Y 446.436,Z 593.355,A -85,B 0,C 180,E1 -8896.107,E2 -8896.107} C_VEL
LIN {X 0,Y 443.278,Z 601.564,A -85,B 0,C 180,E1 -8896.692,E2 -8896.692} C_VEL
LIN {X 0,Y 442.218,Z 606.28,A -85,B 0,C 180,E1 -8897.122,E2 -8897.122} C_VEL
LIN {X 0,Y 441.667,Z 616.352,A -85,B 0,C 180,E1 -8898.295,E2 -8898.295} C_VEL
LIN {X 0,Y 441.137,Z 625.841,A -85,B 0,C 180,E1 -8899.675,E2 -8899.675} C_VEL
LIN {X 0,Y 440.583,Z 633.529,A -85,B 0,C 180,E1 -8901.076,E2 -8901.076} C_VEL
LIN {X 0,Y 440.212,Z 639.285,A -85,B 0,C 180,E1 -8902.384,E2 -8902.384} C_VEL
LIN {X 0,Y 440.004,Z 643.558,A -85,B 0,C 180,E1 -8903.581,E2 -8903.581} C_VEL
LIN {X 0,Y 439.625,Z 647.452,A -85,B 0,C 180,E1 -8904.956,E2 -8904.956} C_VEL
LIN {X 0,Y 439.388,Z 650.319,A -85,B 0,C 180,E1 -8906.332,E2 -8906.332} C_VEL
LIN {X 0,Y 439.414,Z 651.676,A -85,B 0,C 180,E1 -8907.25,E2 -8907.25} C_VEL
LIN {X 0,Y 439.269,Z 652.662,A -85,B 0,C 180,E1 -8908.166,E2 -8908.166} C_VEL
LIN {X 0,Y 439.348,Z 653.246,A -85,B 0,C 180,E1 -8909.083,E2 -8909.083} C_VEL
LIN {X 0,Y 439.332,Z 653.477,A -85,B 0,C 180,E1 -8910,E2 -8910} C_VEL
LIN {X 0,Y 439.348,Z 653.294,A -85,B 0,C 180,E1 -8910.917,E2 -8910.917} C_VEL
LIN {X 0,Y 439.269,Z 652.74,A -85,B 0,C 180,E1 -8911.834,E2 -8911.834} C_VEL
LIN {X 0,Y 439.412,Z 651.785,A -85,B 0,C 180,E1 -8912.75,E2 -8912.75} C_VEL
LIN {X 0,Y 439.381,Z 650.477,A -85,B 0,C 180,E1 -8913.668,E2 -8913.668} C_VEL
LIN {X 0,Y 439.618,Z 647.668,A -85,B 0,C 180,E1 -8915.044,E2 -8915.044} C_VEL
LIN {X 0,Y 439.987,Z 643.849,A -85,B 0,C 180,E1 -8916.42,E2 -8916.42} C_VEL
LIN {X 0,Y 440.197,Z 638.775,A -85,B 0,C 180,E1 -8917.846,E2 -8917.846} C_VEL
LIN {X 0,Y 440.637,Z 632.755,A -85,B 0,C 180,E1 -8919.177,E2 -8919.177} C_VEL
LIN {X 0,Y 441.218,Z 624.98,A -85,B 0,C 180,E1 -8920.555,E2 -8920.555} C_VEL
LIN {X 0,Y 441.75,Z 615.315,A -85,B 0,C 180,E1 -8921.936,E2 -8921.936} C_VEL
LIN {X 0,Y 442.298,Z 606.284,A -85,B 0,C 180,E1 -8922.97,E2 -8922.97} C_VEL
LIN {X 0,Y 442.896,Z 595.794,A -85,B 0,C 180,E1 -8923.939,E2 -8923.939} C_VEL
LIN {X 0,Y 443.306,Z 584.299,A -85,B 0,C 180,E1 -8924.789,E2 -8924.789} C_VEL
LIN {X 0,Y 443.696,Z 573.054,A -85,B 0,C 180,E1 -8925.426,E2 -8925.426} C_VEL
LIN {X 0,Y 443.881,Z 559.884,A -85,B 0,C 180,E1 -8925.968,E2 -8925.968} C_VEL
LIN {X 0,Y 443.914,Z 546.158,A -85,B 0,C 180,E1 -8926.32,E2 -8926.32} C_VEL
LIN {X 0,Y 444.329,Z 483.029,A -85,B 0,C 180,E1 -8927.357,E2 -8927.357} C_VEL
LIN {X 0,Y 439.663,Z 470.725,A -85,B 0,C 180,E1 -8927.787,E2 -8927.787} C_VEL
LIN {X 0,Y 439.462,Z 469.84,A -85,B 0,C 180,E1 -8927.959,E2 -8927.959} C_VEL
LIN {X 0,Y 439.392,Z 469.756,A -85,B 0,C 180,E1 -8930.602,E2 -8930.602} C_VEL
LIN {X 0,Y 439.416,Z 469.748,A -85,B 0,C 180,E1 -8934.264,E2 -8934.264} C_VEL
LIN {X 0,Y 439.441,Z 469.725,A -85,B 0,C 180,E1 -8937.632,E2 -8937.632} C_VEL
LIN {X 0,Y 439.361,Z 469.759,A -85,B 0,C 180,E1 -8940.788,E2 -8940.788} C_VEL
LIN {X 0,Y 439.386,Z 469.75,A -85,B 0,C 180,E1 -8944.043,E2 -8944.043} C_VEL
LIN {X 0,Y 439.355,Z 469.749,A -85,B 0,C 180,E1 -8946.888,E2 -8946.888} C_VEL
LIN {X 0,Y 439.404,Z 469.749,A -85,B 0,C 180,E1 -8949.849,E2 -8949.849} C_VEL
LIN {X 0,Y 439.382,Z 469.741,A -85,B 0,C 180,E1 -8952.627,E2 -8952.627} C_VEL
LIN {X 0,Y 439.398,Z 469.755,A -85,B 0,C 180,E1 -8955.27,E2 -8955.27} C_VEL
LIN {X 0,Y 439.383,Z 469.744,A -85,B 0,C 180,E1 -8958.742,E2 -8958.742} C_VEL
LIN {X 0,Y 439.374,Z 469.747,A -85,B 0,C 180,E1 -8961.606,E2 -8961.606} C_VEL
LIN {X 0,Y 439.395,Z 469.752,A -85,B 0,C 180,E1 -8964.843,E2 -8964.843} C_VEL
LIN {X 0,Y 439.368,Z 469.734,A -85,B 0,C 180,E1 -8968.139,E2 -8968.139} C_VEL
LIN {X 0,Y 439.418,Z 469.734,A -85,B 0,C 180,E1 -8971.326,E2 -8971.326} C_VEL
LIN {X 0,Y 439.398,Z 469.748,A -85,B 0,C 180,E1 -8974.415,E2 -8974.415} C_VEL
LIN {X 0,Y 439.357,Z 469.75,A -85,B 0,C 180,E1 -8977.424,E2 -8977.424} C_VEL
LIN {X 0,Y 439.433,Z 469.744,A -85,B 0,C 180,E1 -8980.662,E2 -8980.662} C_VEL
LIN {X 0,Y 439.454,Z 469.733,A -85,B 0,C 180,E1 -8984.224,E2 -8984.224} C_VEL
LIN {X 0,Y 439.475,Z 469.738,A -85,B 0,C 180,E1 -8988.001,E2 -8988.001} C_VEL
LIN {X 0,Y 439.539,Z 469.73,A -85,B 0,C 180,E1 -8991.726,E2 -8991.726} C_VEL
LIN {X 0,Y 439.613,Z 469.72,A -85,B 0,C 180,E1 -8994.496,E2 -8994.496} C_VEL
LIN {X 0,Y 439.627,Z 469.713,A -85,B 0,C 180,E1 -8998.168,E2 -8998.168} C_VEL
LIN {X 0,Y 439.755,Z 469.703,A -85,B 0,C 180,E1 -9000,E2 -9000} C_VEL
LIN {X 0,Y 439.648,Z 469.713,A -85,B 0,C 180,E1 -9002.749,E2 -9002.749} C_VEL
LIN {X 0,Y 439.612,Z 469.719,A -85,B 0,C 180,E1 -9006.425,E2 -9006.425} C_VEL
LIN {X 0,Y 439.491,Z 469.739,A -85,B 0,C 180,E1 -9009.202,E2 -9009.202} C_VEL
LIN {X 0,Y 439.456,Z 469.739,A -85,B 0,C 180,E1 -9012.938,E2 -9012.938} C_VEL
LIN {X 0,Y 439.438,Z 469.738,A -85,B 0,C 180,E1 -9016.349,E2 -9016.349} C_VEL
LIN {X 0,Y 439.394,Z 469.736,A -85,B 0,C 180,E1 -9019.627,E2 -9019.627} C_VEL
LIN {X 0,Y 439.357,Z 469.753,A -85,B 0,C 180,E1 -9022.576,E2 -9022.576} C_VEL
LIN {X 0,Y 439.398,Z 469.744,A -85,B 0,C 180,E1 -9025.585,E2 -9025.585} C_VEL
LIN {X 0,Y 439.418,Z 469.743,A -85,B 0,C 180,E1 -9028.673,E2 -9028.673} C_VEL
LIN {X 0,Y 439.376,Z 469.747,A -85,B 0,C 180,E1 -9032.034,E2 -9032.034} C_VEL
LIN {X 0,Y 439.39,Z 469.751,A -85,B 0,C 180,E1 -9035.341,E2 -9035.341} C_VEL
LIN {X 0,Y 439.384,Z 469.746,A -85,B 0,C 180,E1 -9038.595,E2 -9038.595} C_VEL
LIN {X 0,Y 439.383,Z 469.753,A -85,B 0,C 180,E1 -9041.258,E2 -9041.258} C_VEL
LIN {X 0,Y 439.398,Z 469.736,A -85,B 0,C 180,E1 -9044.73,E2 -9044.73} C_VEL
LIN {X 0,Y 439.409,Z 469.75,A -85,B 0,C 180,E1 -9047.798,E2 -9047.798} C_VEL
LIN {X 0,Y 439.446,Z 469.737,A -85,B 0,C 180,E1 -9050.231,E2 -9050.231} C_VEL
LIN {X 0,Y 439.374,Z 469.746,A -85,B 0,C 180,E1 -9053.714,E2 -9053.714} C_VEL
LIN {X 0,Y 439.371,Z 469.749,A -85,B 0,C 180,E1 -9057.055,E2 -9057.055} C_VEL
LIN {X 0,Y 439.418,Z 469.926,A -85,B 0,C 180,E1 -9058.581,E2 -9058.581} C_VEL
LIN {X 0,Y 442.848,Z 484.78,A -85,B 0,C 180,E1 -9061.037,E2 -9061.037} C_VEL
LIN {X 0,Y 443.82,Z 490.243,A -85,B 0,C 180,E1 -9061.893,E2 -9061.893} C_VEL
LIN {X 0,Y 442.725,Z 511.387,A -85,B 0,C 180,E1 -9064.919,E2 -9064.919} C_VEL
LIN {X 0,Y 441.598,Z 533.471,A -85,B 0,C 180,E1 -9068.038,E2 -9068.038} C_VEL
LIN {X 0,Y 440.545,Z 557.202,A -85,B 0,C 180,E1 -9071.394,E2 -9071.394} C_VEL
LIN {X 0,Y 440.441,Z 560.277,A -85,B 0,C 180,E1 -9071.812,E2 -9071.812} C_VEL
LIN {X 0,Y 443.739,Z 591.411,A -85,B 0,C 180,E1 -9072.487,E2 -9072.487} C_VEL
LIN {X 0,Y 443.003,Z 670.877,A -85,B 0,C 180,E1 -9073.793,E2 -9073.793} C_VEL
LIN {X 0,Y 442.534,Z 684.201,A -85,B 0,C 180,E1 -9074.19,E2 -9074.19} C_VEL
LIN {X 0,Y 441.848,Z 696.424,A -85,B 0,C 180,E1 -9074.726,E2 -9074.726} C_VEL
LIN {X 0,Y 441.247,Z 708.823,A -85,B 0,C 180,E1 -9075.472,E2 -9075.472} C_VEL
LIN {X 0,Y 440.525,Z 720.685,A -85,B 0,C 180,E1 -9076.402,E2 -9076.402} C_VEL
LIN {X 0,Y 440.061,Z 731.169,A -85,B 0,C 180,E1 -9077.432,E2 -9077.432} C_VEL
LIN {X 0,Y 439.488,Z 739.846,A -85,B 0,C 180,E1 -9078.47,E2 -9078.47} C_VEL
LIN {X 0,Y 439.118,Z 747.894,A -85,B 0,C 180,E1 -9079.627,E2 -9079.627} C_VEL
LIN {X 0,Y 438.82,Z 755.781,A -85,B 0,C 180,E1 -9081.017,E2 -9081.017} C_VEL
LIN {X 0,Y 438.704,Z 763.08,A -85,B 0,C 180,E1 -9082.637,E2 -9082.637} C_VEL
LIN {X 0,Y 438.716,Z 767.957,A -85,B 0,C 180,E1 -9084.023,E2 -9084.023} C_VEL
LIN {X 0,Y 438.765,Z 771.693,A -85,B 0,C 180,E1 -9085.406,E2 -9085.406} C_VEL
LIN {X 0,Y 438.793,Z 773.621,A -85,B 0,C 180,E1 -9086.327,E2 -9086.327} C_VEL
LIN {X 0,Y 438.782,Z 775.063,A -85,B 0,C 180,E1 -9087.246,E2 -9087.246} C_VEL
LIN {X 0,Y 438.98,Z 776.749,A -85,B 0,C 180,E1 -9089.083,E2 -9089.083} C_VEL
LIN {X 0,Y 438.986,Z 776.973,A -85,B 0,C 180,E1 -9090,E2 -9090} C_VEL
LIN {X 0,Y 438.98,Z 776.749,A -85,B 0,C 180,E1 -9090.917,E2 -9090.917} C_VEL
LIN {X 0,Y 438.782,Z 775.065,A -85,B 0,C 180,E1 -9092.754,E2 -9092.754} C_VEL
LIN {X 0,Y 438.793,Z 773.622,A -85,B 0,C 180,E1 -9093.673,E2 -9093.673} C_VEL
LIN {X 0,Y 438.737,Z 770.582,A -85,B 0,C 180,E1 -9095.054,E2 -9095.054} C_VEL
LIN {X 0,Y 438.686,Z 765.744,A -85,B 0,C 180,E1 -9096.646,E2 -9096.646} C_VEL
LIN {X 0,Y 438.771,Z 759.132,A -85,B 0,C 180,E1 -9098.288,E2 -9098.288} C_VEL
LIN {X 0,Y 438.96,Z 752.048,A -85,B 0,C 180,E1 -9099.678,E2 -9099.678} C_VEL
LIN {X 0,Y 439.327,Z 743.215,A -85,B 0,C 180,E1 -9101.067,E2 -9101.067} C_VEL
LIN {X 0,Y 439.852,Z 734.203,A -85,B 0,C 180,E1 -9102.222,E2 -9102.222} C_VEL
LIN {X 0,Y 440.323,Z 724.231,A -85,B 0,C 180,E1 -9103.273,E2 -9103.273} C_VEL
LIN {X 0,Y 440.92,Z 713.549,A -85,B 0,C 180,E1 -9104.186,E2 -9104.186} C_VEL
LIN {X 0,Y 441.679,Z 701.565,A -85,B 0,C 180,E1 -9104.985,E2 -9104.985} C_VEL
LIN {X 0,Y 442.288,Z 689.119,A -85,B 0,C 180,E1 -9105.613,E2 -9105.613} C_VEL
LIN {X 0,Y 442.865,Z 676.383,A -85,B 0,C 180,E1 -9106.064,E2 -9106.064} C_VEL
LIN {X 0,Y 443.145,Z 663.072,A -85,B 0,C 180,E1 -9106.35,E2 -9106.35} C_VEL
LIN {X 0,Y 443.657,Z 590.05,A -85,B 0,C 180,E1 -9107.535,E2 -9107.535} C_VEL
LIN {X 0,Y 440.442,Z 560.524,A -85,B 0,C 180,E1 -9108.167,E2 -9108.167} C_VEL
LIN {X 0,Y 441.413,Z 536.849,A -85,B 0,C 180,E1 -9111.481,E2 -9111.481} C_VEL
LIN {X 0,Y 442.622,Z 513.181,A -85,B 0,C 180,E1 -9114.823,E2 -9114.823} C_VEL
LIN {X 0,Y 443.816,Z 491.933,A -85,B 0,C 180,E1 -9117.851,E2 -9117.851} C_VEL
LIN {X 0,Y 443.351,Z 487.029,A -85,B 0,C 180,E1 -9118.596,E2 -9118.596} C_VEL
LIN {X 0,Y 439.969,Z 472.232,A -85,B 0,C 180,E1 -9121.007,E2 -9121.007} C_VEL
LIN {X 0,Y 439.396,Z 469.852,A -85,B 0,C 180,E1 -9121.454,E2 -9121.454} C_VEL
LIN {X 0,Y 439.385,Z 469.749,A -85,B 0,C 180,E1 -9124.043,E2 -9124.043} C_VEL
LIN {X 0,Y 439.36,Z 469.752,A -85,B 0,C 180,E1 -9127.433,E2 -9127.433} C_VEL
LIN {X 0,Y 439.423,Z 469.738,A -85,B 0,C 180,E1 -9129.852,E2 -9129.852} C_VEL
LIN {X 0,Y 439.4,Z 469.753,A -85,B 0,C 180,E1 -9132.629,E2 -9132.629} C_VEL
LIN {X 0,Y 439.398,Z 469.736,A -85,B 0,C 180,E1 -9135.27,E2 -9135.27} C_VEL
LIN {X 0,Y 439.383,Z 469.753,A -85,B 0,C 180,E1 -9138.742,E2 -9138.742} C_VEL
LIN {X 0,Y 439.38,Z 469.747,A -85,B 0,C 180,E1 -9141.605,E2 -9141.605} C_VEL
LIN {X 0,Y 439.395,Z 469.748,A -85,B 0,C 180,E1 -9144.844,E2 -9144.844} C_VEL
LIN {X 0,Y 439.369,Z 469.75,A -85,B 0,C 180,E1 -9148.139,E2 -9148.139} C_VEL
LIN {X 0,Y 439.418,Z 469.742,A -85,B 0,C 180,E1 -9151.327,E2 -9151.327} C_VEL
LIN {X 0,Y 439.398,Z 469.744,A -85,B 0,C 180,E1 -9154.415,E2 -9154.415} C_VEL
LIN {X 0,Y 439.357,Z 469.753,A -85,B 0,C 180,E1 -9157.424,E2 -9157.424} C_VEL
LIN {X 0,Y 439.433,Z 469.729,A -85,B 0,C 180,E1 -9160.662,E2 -9160.662} C_VEL
LIN {X 0,Y 439.453,Z 469.741,A -85,B 0,C 180,E1 -9164.224,E2 -9164.224} C_VEL
LIN {X 0,Y 439.475,Z 469.737,A -85,B 0,C 180,E1 -9168.001,E2 -9168.001} C_VEL
LIN {X 0,Y 439.539,Z 469.73,A -85,B 0,C 180,E1 -9171.726,E2 -9171.726} C_VEL
LIN {X 0,Y 439.618,Z 469.719,A -85,B 0,C 180,E1 -9174.496,E2 -9174.496} C_VEL
LIN {X 0,Y 439.627,Z 469.72,A -85,B 0,C 180,E1 -9178.168,E2 -9178.168} C_VEL
LIN {X 0,Y 439.755,Z 469.704,A -85,B 0,C 180,E1 -9180,E2 -9180} C_VEL
LIN {X 0,Y 439.648,Z 469.713,A -85,B 0,C 180,E1 -9182.749,E2 -9182.749} C_VEL
LIN {X 0,Y 439.613,Z 469.725,A -85,B 0,C 180,E1 -9186.425,E2 -9186.425} C_VEL
LIN {X 0,Y 439.492,Z 469.728,A -85,B 0,C 180,E1 -9189.202,E2 -9189.202} C_VEL
LIN {X 0,Y 439.457,Z 469.745,A -85,B 0,C 180,E1 -9192.938,E2 -9192.938} C_VEL
LIN {X 0,Y 439.439,Z 469.738,A -85,B 0,C 180,E1 -9196.349,E2 -9196.349} C_VEL
LIN {X 0,Y 439.394,Z 469.748,A -85,B 0,C 180,E1 -9199.627,E2 -9199.627} C_VEL
LIN {X 0,Y 439.357,Z 469.75,A -85,B 0,C 180,E1 -9202.576,E2 -9202.576} C_VEL
LIN {X 0,Y 439.398,Z 469.748,A -85,B 0,C 180,E1 -9205.585,E2 -9205.585} C_VEL
LIN {X 0,Y 439.418,Z 469.735,A -85,B 0,C 180,E1 -9208.674,E2 -9208.674} C_VEL
LIN {X 0,Y 439.368,Z 469.733,A -85,B 0,C 180,E1 -9211.861,E2 -9211.861} C_VEL
LIN {X 0,Y 439.395,Z 469.753,A -85,B 0,C 180,E1 -9215.157,E2 -9215.157} C_VEL
LIN {X 0,Y 439.375,Z 469.744,A -85,B 0,C 180,E1 -9218.596,E2 -9218.596} C_VEL
LIN {X 0,Y 439.383,Z 469.741,A -85,B 0,C 180,E1 -9221.258,E2 -9221.258} C_VEL
LIN {X 0,Y 439.398,Z 469.753,A -85,B 0,C 180,E1 -9224.73,E2 -9224.73} C_VEL
LIN {X 0,Y 439.395,Z 469.739,A -85,B 0,C 180,E1 -9227.797,E2 -9227.797} C_VEL
LIN {X 0,Y 439.435,Z 469.744,A -85,B 0,C 180,E1 -9230.229,E2 -9230.229} C_VEL
LIN {X 0,Y 439.375,Z 469.731,A -85,B 0,C 180,E1 -9233.714,E2 -9233.714} C_VEL
LIN {X 0,Y 439.371,Z 469.731,A -85,B 0,C 180,E1 -9237.055,E2 -9237.055} C_VEL
LIN {X 0,Y 439.382,Z 469.753,A -85,B 0,C 180,E1 -9240.275,E2 -9240.275} C_VEL
LIN {X 0,Y 439.429,Z 469.727,A -85,B 0,C 180,E1 -9243.397,E2 -9243.397} C_VEL
LIN {X 0,Y 439.388,Z 469.751,A -85,B 0,C 180,E1 -9246.43,E2 -9246.43} C_VEL
LIN {X 0,Y 439.391,Z 469.754,A -85,B 0,C 180,E1 -9249.398,E2 -9249.398} C_VEL
LIN {X 0,Y 439.477,Z 469.874,A -85,B 0,C 180,E1 -9252.162,E2 -9252.162} C_VEL
LIN {X 0,Y 439.701,Z 470.916,A -85,B 0,C 180,E1 -9252.321,E2 -9252.321} C_VEL
LIN {X 0,Y 444.422,Z 483.287,A -85,B 0,C 180,E1 -9252.747,E2 -9252.747} C_VEL
LIN {X 0,Y 443.957,Z 550.295,A -85,B 0,C 180,E1 -9253.858,E2 -9253.858} C_VEL
LIN {X 0,Y 443.887,Z 563.01,A -85,B 0,C 180,E1 -9254.239,E2 -9254.239} C_VEL
LIN {X 0,Y 443.575,Z 575.387,A -85,B 0,C 180,E1 -9254.787,E2 -9254.787} C_VEL
LIN {X 0,Y 443.262,Z 586.641,A -85,B 0,C 180,E1 -9255.463,E2 -9255.463} C_VEL
LIN {X 0,Y 442.74,Z 596.71,A -85,B 0,C 180,E1 -9256.225,E2 -9256.225} C_VEL
LIN {X 0,Y 442.218,Z 606.28,A -85,B 0,C 180,E1 -9257.122,E2 -9257.122} C_VEL
LIN {X 0,Y 441.164,Z 610.93,A -85,B 0,C 180,E1 -9257.58,E2 -9257.58} C_VEL
LIN {X 0,Y 437.969,Z 618.228,A -85,B 0,C 180,E1 -9258.354,E2 -9258.354} C_VEL
LIN {X 0,Y 434.91,Z 624.922,A -85,B 0,C 180,E1 -9259.22,E2 -9259.22} C_VEL
LIN {X 0,Y 434.074,Z 628.62,A -85,B 0,C 180,E1 -9259.815,E2 -9259.815} C_VEL
LIN {X 0,Y 433.559,Z 635.715,A -85,B 0,C 180,E1 -9261.189,E2 -9261.189} C_VEL
LIN {X 0,Y 433.205,Z 641.331,A -85,B 0,C 180,E1 -9262.543,E2 -9262.543} C_VEL
LIN {X 0,Y 432.805,Z 645.952,A -85,B 0,C 180,E1 -9263.941,E2 -9263.941} C_VEL
LIN {X 0,Y 432.519,Z 649.484,A -85,B 0,C 180,E1 -9265.34,E2 -9265.34} C_VEL
LIN {X 0,Y 432.372,Z 651.309,A -85,B 0,C 180,E1 -9266.272,E2 -9266.272} C_VEL
LIN {X 0,Y 432.396,Z 652.665,A -85,B 0,C 180,E1 -9267.205,E2 -9267.205} C_VEL
LIN {X 0,Y 432.247,Z 653.65,A -85,B 0,C 180,E1 -9268.137,E2 -9268.137} C_VEL
LIN {X 0,Y 432.326,Z 654.234,A -85,B 0,C 180,E1 -9269.069,E2 -9269.069} C_VEL
LIN {X 0,Y 432.309,Z 654.465,A -85,B 0,C 180,E1 -9270,E2 -9270} C_VEL
LIN {X 0,Y 432.326,Z 654.281,A -85,B 0,C 180,E1 -9270.931,E2 -9270.931} C_VEL
LIN {X 0,Y 432.247,Z 653.727,A -85,B 0,C 180,E1 -9271.863,E2 -9271.863} C_VEL
LIN {X 0,Y 432.394,Z 652.772,A -85,B 0,C 180,E1 -9272.795,E2 -9272.795} C_VEL
LIN {X 0,Y 432.364,Z 651.465,A -85,B 0,C 180,E1 -9273.728,E2 -9273.728} C_VEL
LIN {X 0,Y 432.616,Z 648.656,A -85,B 0,C 180,E1 -9275.126,E2 -9275.126} C_VEL
LIN {X 0,Y 433.004,Z 644.836,A -85,B 0,C 180,E1 -9276.524,E2 -9276.524} C_VEL
LIN {X 0,Y 433.236,Z 639.762,A -85,B 0,C 180,E1 -9277.972,E2 -9277.972} C_VEL
LIN {X 0,Y 433.702,Z 633.741,A -85,B 0,C 180,E1 -9279.325,E2 -9279.325} C_VEL
LIN {X 0,Y 434.31,Z 625.965,A -85,B 0,C 180,E1 -9280.725,E2 -9280.725} C_VEL
LIN {X 0,Y 434.875,Z 616.299,A -85,B 0,C 180,E1 -9282.127,E2 -9282.127} C_VEL
LIN {X 0,Y 435.452,Z 607.268,A -85,B 0,C 180,E1 -9283.177,E2 -9283.177} C_VEL
LIN {X 0,Y 436.078,Z 596.776,A -85,B 0,C 180,E1 -9284.162,E2 -9284.162} C_VEL
LIN {X 0,Y 436.535,Z 585.124,A -85,B 0,C 180,E1 -9285.034,E2 -9285.034} C_VEL
LIN {X 0,Y 436.923,Z 573.701,A -85,B 0,C 180,E1 -9285.689,E2 -9285.689} C_VEL
LIN {X 0,Y 437.115,Z 560.861,A -85,B 0,C 180,E1 -9286.221,E2 -9286.221} C_VEL
LIN {X 0,Y 437.152,Z 547.126,A -85,B 0,C 180,E1 -9286.58,E2 -9286.58} C_VEL
LIN {X 0,Y 437.602,Z 484.636,A -85,B 0,C 180,E1 -9287.621,E2 -9287.621} C_VEL
LIN {X 0,Y 432.622,Z 471.683,A -85,B 0,C 180,E1 -9288.083,E2 -9288.083} C_VEL
LIN {X 0,Y 432.403,Z 470.724,A -85,B 0,C 180,E1 -9288.263,E2 -9288.263} C_VEL
LIN {X 0,Y 432.353,Z 470.625,A -85,B 0,C 180,E1 -9290.953,E2 -9290.953} C_VEL
LIN {X 0,Y 432.384,Z 470.626,A -85,B 0,C 180,E1 -9294.463,E2 -9294.463} C_VEL
LIN {X 0,Y 432.391,Z 470.6,A -85,B 0,C 180,E1 -9297.071,E2 -9297.071} C_VEL
LIN {X 0,Y 432.347,Z 470.63,A -85,B 0,C 180,E1 -9300.51,E2 -9300.51} C_VEL
LIN {X 0,Y 432.358,Z 470.626,A -85,B 0,C 180,E1 -9304.003,E2 -9304.003} C_VEL
LIN {X 0,Y 432.33,Z 470.624,A -85,B 0,C 180,E1 -9307.198,E2 -9307.198} C_VEL
LIN {X 0,Y 432.334,Z 470.629,A -85,B 0,C 180,E1 -9310.179,E2 -9310.179} C_VEL
LIN {X 0,Y 432.32,Z 470.621,A -85,B 0,C 180,E1 -9313.059,E2 -9313.059} C_VEL
LIN {X 0,Y 432.329,Z 470.632,A -85,B 0,C 180,E1 -9315.664,E2 -9315.664} C_VEL
LIN {X 0,Y 432.328,Z 470.624,A -85,B 0,C 180,E1 -9318.397,E2 -9318.397} C_VEL
LIN {X 0,Y 432.338,Z 470.623,A -85,B 0,C 180,E1 -9321.85,E2 -9321.85} C_VEL
LIN {X 0,Y 432.335,Z 470.63,A -85,B 0,C 180,E1 -9325.322,E2 -9325.322} C_VEL
LIN {X 0,Y 432.317,Z 470.609,A -85,B 0,C 180,E1 -9328.653,E2 -9328.653} C_VEL
LIN {X 0,Y 432.374,Z 470.612,A -85,B 0,C 180,E1 -9331.368,E2 -9331.368} C_VEL
LIN {X 0,Y 432.357,Z 470.625,A -85,B 0,C 180,E1 -9333.967,E2 -9333.967} C_VEL
LIN {X 0,Y 432.311,Z 470.63,A -85,B 0,C 180,E1 -9337.035,E2 -9337.035} C_VEL
LIN {X 0,Y 432.379,Z 470.622,A -85,B 0,C 180,E1 -9340.514,E2 -9340.514} C_VEL
LIN {X 0,Y 432.422,Z 470.61,A -85,B 0,C 180,E1 -9343.961,E2 -9343.961} C_VEL
LIN {X 0,Y 432.451,Z 470.614,A -85,B 0,C 180,E1 -9347.803,E2 -9347.803} C_VEL
LIN {X 0,Y 432.483,Z 470.608,A -85,B 0,C 180,E1 -9351.59,E2 -9351.59} C_VEL
LIN {X 0,Y 432.589,Z 470.594,A -85,B 0,C 180,E1 -9354.406,E2 -9354.406} C_VEL
LIN {X 0,Y 432.597,Z 470.588,A -85,B 0,C 180,E1 -9358.138,E2 -9358.138} C_VEL
LIN {X 0,Y 432.725,Z 470.579,A -85,B 0,C 180,E1 -9360,E2 -9360} C_VEL
LIN {X 0,Y 432.597,Z 470.591,A -85,B 0,C 180,E1 -9362.794,E2 -9362.794} C_VEL
LIN {X 0,Y 432.566,Z 470.597,A -85,B 0,C 180,E1 -9366.53,E2 -9366.53} C_VEL
LIN {X 0,Y 432.434,Z 470.618,A -85,B 0,C 180,E1 -9369.353,E2 -9369.353} C_VEL
LIN {X 0,Y 432.422,Z 470.614,A -85,B 0,C 180,E1 -9372.804,E2 -9372.804} C_VEL
LIN {X 0,Y 432.404,Z 470.614,A -85,B 0,C 180,E1 -9376.479,E2 -9376.479} C_VEL
LIN {X 0,Y 432.331,Z 470.62,A -85,B 0,C 180,E1 -9379.961,E2 -9379.961} C_VEL
LIN {X 0,Y 432.311,Z 470.632,A -85,B 0,C 180,E1 -9382.965,E2 -9382.965} C_VEL
LIN {X 0,Y 432.357,Z 470.614,A -85,B 0,C 180,E1 -9386.033,E2 -9386.033} C_VEL
LIN {X 0,Y 432.346,Z 470.626,A -85,B 0,C 180,E1 -9389.187,E2 -9389.187} C_VEL
LIN {X 0,Y 432.325,Z 470.623,A -85,B 0,C 180,E1 -9392.295,E2 -9392.295} C_VEL
LIN {X 0,Y 432.335,Z 470.626,A -85,B 0,C 180,E1 -9394.678,E2 -9394.678} C_VEL
LIN {X 0,Y 432.342,Z 470.624,A -85,B 0,C 180,E1 -9398.15,E2 -9398.15} C_VEL
LIN {X 0,Y 432.328,Z 470.63,A -85,B 0,C 180,E1 -9401.603,E2 -9401.603} C_VEL
LIN {X 0,Y 432.329,Z 470.612,A -85,B 0,C 180,E1 -9404.348,E2 -9404.348} C_VEL
LIN {X 0,Y 432.362,Z 470.627,A -85,B 0,C 180,E1 -9407.01,E2 -9407.01} C_VEL
LIN {X 0,Y 432.353,Z 470.617,A -85,B 0,C 180,E1 -9409.818,E2 -9409.818} C_VEL
LIN {X 0,Y 432.314,Z 470.628,A -85,B 0,C 180,E1 -9413.024,E2 -9413.024} C_VEL
LIN {X 0,Y 432.358,Z 470.623,A -85,B 0,C 180,E1 -9415.997,E2 -9415.997} C_VEL
LIN {X 0,Y 432.365,Z 470.831,A -85,B 0,C 180,E1 -9418.3,E2 -9418.3} C_VEL
LIN {X 0,Y 435.816,Z 485.683,A -85,B 0,C 180,E1 -9420.801,E2 -9420.801} C_VEL
LIN {X 0,Y 436.966,Z 492.836,A -85,B 0,C 180,E1 -9421.937,E2 -9421.937} C_VEL
LIN {X 0,Y 435.596,Z 515.317,A -85,B 0,C 180,E1 -9425.198,E2 -9425.198} C_VEL
LIN {X 0,Y 434.506,Z 535.919,A -85,B 0,C 180,E1 -9428.16,E2 -9428.16} C_VEL
LIN {X 0,Y 433.465,Z 559.288,A -85,B 0,C 180,E1 -9431.511,E2 -9431.511} C_VEL
LIN {X 0,Y 436.932,Z 591.748,A -85,B 0,C 180,E1 -9432.228,E2 -9432.228} C_VEL
LIN {X 0,Y 436.186,Z 669.89,A -85,B 0,C 180,E1 -9433.533,E2 -9433.533} C_VEL
LIN {X 0,Y 435.671,Z 683.205,A -85,B 0,C 180,E1 -9433.934,E2 -9433.934} C_VEL
LIN {X 0,Y 434.976,Z 695.428,A -85,B 0,C 180,E1 -9434.479,E2 -9434.479} C_VEL
LIN {X 0,Y 434.362,Z 707.826,A -85,B 0,C 180,E1 -9435.237,E2 -9435.237} C_VEL
LIN {X 0,Y 433.681,Z 718.374,A -85,B 0,C 180,E1 -9436.063,E2 -9436.063} C_VEL
LIN {X 0,Y 433.083,Z 729.069,A -85,B 0,C 180,E1 -9437.107,E2 -9437.107} C_VEL
LIN {X 0,Y 432.424,Z 738.834,A -85,B 0,C 180,E1 -9438.279,E2 -9438.279} C_VEL
LIN {X 0,Y 432.056,Z 746.886,A -85,B 0,C 180,E1 -9439.456,E2 -9439.456} C_VEL
LIN {X 0,Y 431.772,Z 754.778,A -85,B 0,C 180,E1 -9440.869,E2 -9440.869} C_VEL
LIN {X 0,Y 431.633,Z 762.079,A -85,B 0,C 180,E1 -9442.516,E2 -9442.516} C_VEL
LIN {X 0,Y 431.654,Z 766.96,A -85,B 0,C 180,E1 -9443.925,E2 -9443.925} C_VEL
LIN {X 0,Y 431.717,Z 770.699,A -85,B 0,C 180,E1 -9445.331,E2 -9445.331} C_VEL
LIN {X 0,Y 431.753,Z 772.629,A -85,B 0,C 180,E1 -9446.267,E2 -9446.267} C_VEL
LIN {X 0,Y 431.737,Z 774.072,A -85,B 0,C 180,E1 -9447.201,E2 -9447.201} C_VEL
LIN {X 0,Y 431.957,Z 775.762,A -85,B 0,C 180,E1 -9449.068,E2 -9449.068} C_VEL
LIN {X 0,Y 431.966,Z 775.986,A -85,B 0,C 180,E1 -9450,E2 -9450} C_VEL
LIN {X 0,Y 431.957,Z 775.761,A -85,B 0,C 180,E1 -9450.932,E2 -9450.932} C_VEL
LIN {X 0,Y 431.738,Z 774.073,A -85,B 0,C 180,E1 -9452.799,E2 -9452.799} C_VEL
LIN {X 0,Y 431.752,Z 772.63,A -85,B 0,C 180,E1 -9453.733,E2 -9453.733} C_VEL
LIN {X 0,Y 431.673,Z 769.584,A -85,B 0,C 180,E1 -9455.137,E2 -9455.137} C_VEL
LIN {X 0,Y 431.612,Z 765.121,A -85,B 0,C 180,E1 -9456.649,E2 -9456.649} C_VEL
LIN {X 0,Y 431.689,Z 759.168,A -85,B 0,C 180,E1 -9458.19,E2 -9458.19} C_VEL
LIN {X 0,Y 431.861,Z 752.307,A -85,B 0,C 180,E1 -9459.602,E2 -9459.602} C_VEL
LIN {X 0,Y 432.234,Z 743.833,A -85,B 0,C 180,E1 -9461.014,E2 -9461.014} C_VEL
LIN {X 0,Y 432.707,Z 735.173,A -85,B 0,C 180,E1 -9462.189,E2 -9462.189} C_VEL
LIN {X 0,Y 433.26,Z 724.743,A -85,B 0,C 180,E1 -9463.34,E2 -9463.34} C_VEL
LIN {X 0,Y 433.896,Z 713.985,A -85,B 0,C 180,E1 -9464.3,E2 -9464.3} C_VEL
LIN {X 0,Y 434.68,Z 702.504,A -85,B 0,C 180,E1 -9465.112,E2 -9465.112} C_VEL
LIN {X 0,Y 435.287,Z 690.726,A -85,B 0,C 180,E1 -9465.75,E2 -9465.75} C_VEL
LIN {X 0,Y 435.932,Z 677.207,A -85,B 0,C 180,E1 -9466.267,E2 -9466.267} C_VEL
LIN {X 0,Y 436.315,Z 663.845,A -85,B 0,C 180,E1 -9466.583,E2 -9466.583} C_VEL
LIN {X 0,Y 436.785,Z 590.187,A -85,B 0,C 180,E1 -9467.801,E2 -9467.801} C_VEL
LIN {X 0,Y 433.449,Z 559.543,A -85,B 0,C 180,E1 -9468.468,E2 -9468.468} C_VEL
LIN {X 0,Y 434.415,Z 537.587,A -85,B 0,C 180,E1 -9471.595,E2 -9471.595} C_VEL
LIN {X 0,Y 435.696,Z 514.072,A -85,B 0,C 180,E1 -9474.975,E2 -9474.975} C_VEL
LIN {X 0,Y 436.944,Z 492.787,A -85,B 0,C 180,E1 -9478.064,E2 -9478.064} C_VEL
LIN {X 0,Y 436.228,Z 487.442,A -85,B 0,C 180,E1 -9478.902,E2 -9478.902} C_VEL
LIN {X 0,Y 432.913,Z 473.054,A -85,B 0,C 180,E1 -9481.297,E2 -9481.297} C_VEL
LIN {X 0,Y 432.354,Z 470.719,A -85,B 0,C 180,E1 -9481.752,E2 -9481.752} C_VEL
LIN {X 0,Y 432.338,Z 470.634,A -85,B 0,C 180,E1 -9484.676,E2 -9484.676} C_VEL
LIN {X 0,Y 432.348,Z 470.633,A -85,B 0,C 180,E1 -9488.148,E2 -9488.148} C_VEL
LIN {X 0,Y 432.37,Z 470.62,A -85,B 0,C 180,E1 -9491.607,E2 -9491.607} C_VEL
LIN {X 0,Y 432.374,Z 470.618,A -85,B 0,C 180,E1 -9494.341,E2 -9494.341} C_VEL
LIN {X 0,Y 432.328,Z 470.627,A -85,B 0,C 180,E1 -9498.202,E2 -9498.202} C_VEL
LIN {X 0,Y 432.347,Z 470.622,A -85,B 0,C 180,E1 -9501.283,E2 -9501.283} C_VEL
LIN {X 0,Y 432.34,Z 470.633,A -85,B 0,C 180,E1 -9504.367,E2 -9504.367} C_VEL
LIN {X 0,Y 432.317,Z 470.624,A -85,B 0,C 180,E1 -9507.556,E2 -9507.556} C_VEL
LIN {X 0,Y 432.388,Z 470.623,A -85,B 0,C 180,E1 -9509.743,E2 -9509.743} C_VEL
LIN {X 0,Y 432.393,Z 470.607,A -85,B 0,C 180,E1 -9513.372,E2 -9513.372} C_VEL
LIN {X 0,Y 432.364,Z 470.625,A -85,B 0,C 180,E1 -9516.023,E2 -9516.023} C_VEL
LIN {X 0,Y 432.342,Z 470.62,A -85,B 0,C 180,E1 -9519.046,E2 -9519.046} C_VEL
LIN {X 0,Y 432.369,Z 470.608,A -85,B 0,C 180,E1 -9522.011,E2 -9522.011} C_VEL
LIN {X 0,Y 432.386,Z 470.624,A -85,B 0,C 180,E1 -9524.926,E2 -9524.926} C_VEL
LIN {X 0,Y 432.45,Z 470.611,A -85,B 0,C 180,E1 -9527.803,E2 -9527.803} C_VEL
LIN {X 0,Y 432.483,Z 470.609,A -85,B 0,C 180,E1 -9531.59,E2 -9531.59} C_VEL
LIN {X 0,Y 432.594,Z 470.596,A -85,B 0,C 180,E1 -9534.406,E2 -9534.406} C_VEL
LIN {X 0,Y 432.597,Z 470.595,A -85,B 0,C 180,E1 -9538.138,E2 -9538.138} C_VEL
LIN {X 0,Y 432.725,Z 470.58,A -85,B 0,C 180,E1 -9540,E2 -9540} C_VEL
LIN {X 0,Y 432.597,Z 470.59,A -85,B 0,C 180,E1 -9542.794,E2 -9542.794} C_VEL
LIN {X 0,Y 432.567,Z 470.604,A -85,B 0,C 180,E1 -9546.53,E2 -9546.53} C_VEL
LIN {X 0,Y 432.435,Z 470.606,A -85,B 0,C 180,E1 -9549.353,E2 -9549.353} C_VEL
LIN {X 0,Y 432.422,Z 470.623,A -85,B 0,C 180,E1 -9552.804,E2 -9552.804} C_VEL
LIN {X 0,Y 432.404,Z 470.614,A -85,B 0,C 180,E1 -9556.479,E2 -9556.479} C_VEL
LIN {X 0,Y 432.331,Z 470.628,A -85,B 0,C 180,E1 -9559.961,E2 -9559.961} C_VEL
LIN {X 0,Y 432.311,Z 470.63,A -85,B 0,C 180,E1 -9562.965,E2 -9562.965} C_VEL
LIN {X 0,Y 432.358,Z 470.625,A -85,B 0,C 180,E1 -9566.033,E2 -9566.033} C_VEL
LIN {X 0,Y 432.345,Z 470.608,A -85,B 0,C 180,E1 -9569.187,E2 -9569.187} C_VEL
LIN {X 0,Y 432.319,Z 470.612,A -85,B 0,C 180,E1 -9572.294,E2 -9572.294} C_VEL
LIN {X 0,Y 432.335,Z 470.629,A -85,B 0,C 180,E1 -9574.678,E2 -9574.678} C_VEL
LIN {X 0,Y 432.338,Z 470.622,A -85,B 0,C 180,E1 -9578.15,E2 -9578.15} C_VEL
LIN {X 0,Y 432.328,Z 470.624,A -85,B 0,C 180,E1 -9581.603,E2 -9581.603} C_VEL
LIN {X 0,Y 432.33,Z 470.63,A -85,B 0,C 180,E1 -9584.348,E2 -9584.348} C_VEL
LIN {X 0,Y 432.321,Z 470.62,A -85,B 0,C 180,E1 -9587.016,E2 -9587.016} C_VEL
LIN {X 0,Y 432.34,Z 470.628,A -85,B 0,C 180,E1 -9589.82,E2 -9589.82} C_VEL
LIN {X 0,Y 432.314,Z 470.617,A -85,B 0,C 180,E1 -9593.024,E2 -9593.024} C_VEL
LIN {X 0,Y 432.358,Z 470.589,A -85,B 0,C 180,E1 -9595.997,E2 -9595.997} C_VEL
LIN {X 0,Y 432.347,Z 470.632,A -85,B 0,C 180,E1 -9599.49,E2 -9599.49} C_VEL
LIN {X 0,Y 432.391,Z 470.601,A -85,B 0,C 180,E1 -9602.929,E2 -9602.929} C_VEL
LIN {X 0,Y 432.372,Z 470.625,A -85,B 0,C 180,E1 -9606.024,E2 -9606.024} C_VEL
LIN {X 0,Y 432.352,Z 470.625,A -85,B 0,C 180,E1 -9609.047,E2 -9609.047} C_VEL
LIN {X 0,Y 432.405,Z 470.69,A -85,B 0,C 180,E1 -9611.829,E2 -9611.829} C_VEL
LIN {X 0,Y 432.594,Z 471.577,A -85,B 0,C 180,E1 -9612.006,E2 -9612.006} C_VEL
LIN {X 0,Y 437.598,Z 484.632,A -85,B 0,C 180,E1 -9612.475,E2 -9612.475} C_VEL
LIN {X 0,Y 437.216,Z 551.303,A -85,B 0,C 180,E1 -9613.602,E2 -9613.602} C_VEL
LIN {X 0,Y 437.111,Z 564.012,A -85,B 0,C 180,E1 -9613.988,E2 -9613.988} C_VEL
LIN {X 0,Y 436.794,Z 576.384,A -85,B 0,C 180,E1 -9614.545,E2 -9614.545} C_VEL
LIN {X 0,Y 436.438,Z 588.732,A -85,B 0,C 180,E1 -9615.307,E2 -9615.307} C_VEL
LIN {X 0,Y 435.793,Z 600.318,A -85,B 0,C 180,E1 -9616.239,E2 -9616.239} C_VEL
LIN {X 0,Y 435.206,Z 610.656,A -85,B 0,C 180,E1 -9617.29,E2 -9617.29} C_VEL
LIN {X 0,Y 434.678,Z 619.088,A -85,B 0,C 180,E1 -9618.34,E2 -9618.34} C_VEL
LIN {X 0,Y 434.225,Z 626.832,A -85,B 0,C 180,E1 -9619.509,E2 -9619.509} C_VEL
LIN {X 0,Y 434.074,Z 628.62,A -85,B 0,C 180,E1 -9619.815,E2 -9619.815} C_VEL
LIN {X 0,Y 433.249,Z 631.077,A -85,B 0,C 180,E1 -9620.22,E2 -9620.22} C_VEL
LIN {X 0,Y 427.093,Z 638.504,A -85,B 0,C 180,E1 -9621.48,E2 -9621.48} C_VEL
LIN {X 0,Y 426.315,Z 640.482,A -85,B 0,C 180,E1 -9621.932,E2 -9621.932} C_VEL
LIN {X 0,Y 426.042,Z 645.537,A -85,B 0,C 180,E1 -9623.369,E2 -9623.369} C_VEL
LIN {X 0,Y 425.622,Z 649.431,A -85,B 0,C 180,E1 -9624.789,E2 -9624.789} C_VEL
LIN {X 0,Y 425.356,Z 652.298,A -85,B 0,C 180,E1 -9626.211,E2 -9626.211} C_VEL
LIN {X 0,Y 425.378,Z 653.653,A -85,B 0,C 180,E1 -9627.159,E2 -9627.159} C_VEL
LIN {X 0,Y 425.225,Z 654.638,A -85,B 0,C 180,E1 -9628.106,E2 -9628.106} C_VEL
LIN {X 0,Y 425.303,Z 655.222,A -85,B 0,C 180,E1 -9629.053,E2 -9629.053} C_VEL
LIN {X 0,Y 425.286,Z 655.452,A -85,B 0,C 180,E1 -9630,E2 -9630} C_VEL
LIN {X 0,Y 425.303,Z 655.268,A -85,B 0,C 180,E1 -9630.947,E2 -9630.947} C_VEL
LIN {X 0,Y 425.225,Z 654.715,A -85,B 0,C 180,E1 -9631.894,E2 -9631.894} C_VEL
LIN {X 0,Y 425.375,Z 653.76,A -85,B 0,C 180,E1 -9632.841,E2 -9632.841} C_VEL
LIN {X 0,Y 425.349,Z 652.453,A -85,B 0,C 180,E1 -9633.789,E2 -9633.789} C_VEL
LIN {X 0,Y 425.614,Z 649.643,A -85,B 0,C 180,E1 -9635.211,E2 -9635.211} C_VEL
LIN {X 0,Y 426.023,Z 645.822,A -85,B 0,C 180,E1 -9636.631,E2 -9636.631} C_VEL
LIN {X 0,Y 426.277,Z 640.749,A -85,B 0,C 180,E1 -9638.103,E2 -9638.103} C_VEL
LIN {X 0,Y 426.77,Z 634.727,A -85,B 0,C 180,E1 -9639.478,E2 -9639.478} C_VEL
LIN {X 0,Y 427.407,Z 626.951,A -85,B 0,C 180,E1 -9640.9,E2 -9640.9} C_VEL
LIN {X 0,Y 428.005,Z 617.285,A -85,B 0,C 180,E1 -9642.325,E2 -9642.325} C_VEL
LIN {X 0,Y 428.612,Z 608.252,A -85,B 0,C 180,E1 -9643.391,E2 -9643.391} C_VEL
LIN {X 0,Y 429.267,Z 597.759,A -85,B 0,C 180,E1 -9644.391,E2 -9644.391} C_VEL
LIN {X 0,Y 429.749,Z 586.106,A -85,B 0,C 180,E1 -9645.277,E2 -9645.277} C_VEL
LIN {X 0,Y 430.154,Z 574.681,A -85,B 0,C 180,E1 -9645.943,E2 -9645.943} C_VEL
LIN {X 0,Y 430.367,Z 561.836,A -85,B 0,C 180,E1 -9646.483,E2 -9646.483} C_VEL
LIN {X 0,Y 430.393,Z 548.096,A -85,B 0,C 180,E1 -9646.848,E2 -9646.848} C_VEL
LIN {X 0,Y 430.85,Z 486.201,A -85,B 0,C 180,E1 -9647.896,E2 -9647.896} C_VEL
LIN {X 0,Y 425.533,Z 472.351,A -85,B 0,C 180,E1 -9648.415,E2 -9648.415} C_VEL
LIN {X 0,Y 425.373,Z 471.558,A -85,B 0,C 180,E1 -9648.607,E2 -9648.607} C_VEL
LIN {X 0,Y 425.289,Z 471.491,A -85,B 0,C 180,E1 -9652.338,E2 -9652.338} C_VEL
LIN {X 0,Y 425.296,Z 471.502,A -85,B 0,C 180,E1 -9655.445,E2 -9655.445} C_VEL
LIN {X 0,Y 425.331,Z 471.489,A -85,B 0,C 180,E1 -9658.631,E2 -9658.631} C_VEL
LIN {X 0,Y 425.264,Z 471.505,A -85,B 0,C 180,E1 -9661.926,E2 -9661.926} C_VEL
LIN {X 0,Y 425.299,Z 471.505,A -85,B 0,C 180,E1 -9665.335,E2 -9665.335} C_VEL
LIN {X 0,Y 425.298,Z 471.509,A -85,B 0,C 180,E1 -9669.043,E2 -9669.043} C_VEL
LIN {X 0,Y 425.275,Z 471.497,A -85,B 0,C 180,E1 -9672.652,E2 -9672.652} C_VEL
LIN {X 0,Y 425.257,Z 471.511,A -85,B 0,C 180,E1 -9676.043,E2 -9676.043} C_VEL
LIN {X 0,Y 425.27,Z 471.502,A -85,B 0,C 180,E1 -9678.621,E2 -9678.621} C_VEL
LIN {X 0,Y 425.295,Z 471.489,A -85,B 0,C 180,E1 -9681.101,E2 -9681.101} C_VEL
LIN {X 0,Y 425.295,Z 471.507,A -85,B 0,C 180,E1 -9684.663,E2 -9684.663} C_VEL
LIN {X 0,Y 425.26,Z 471.49,A -85,B 0,C 180,E1 -9688.072,E2 -9688.072} C_VEL
LIN {X 0,Y 425.331,Z 471.488,A -85,B 0,C 180,E1 -9691.368,E2 -9691.368} C_VEL
LIN {X 0,Y 425.288,Z 471.506,A -85,B 0,C 180,E1 -9694.554,E2 -9694.554} C_VEL
LIN {X 0,Y 425.28,Z 471.503,A -85,B 0,C 180,E1 -9697.661,E2 -9697.661} C_VEL
LIN {X 0,Y 425.354,Z 471.499,A -85,B 0,C 180,E1 -9700.704,E2 -9700.704} C_VEL
LIN {X 0,Y 425.38,Z 471.488,A -85,B 0,C 180,E1 -9703.688,E2 -9703.688} C_VEL
LIN {X 0,Y 425.403,Z 471.494,A -85,B 0,C 180,E1 -9707.598,E2 -9707.598} C_VEL
LIN {X 0,Y 425.434,Z 471.484,A -85,B 0,C 180,E1 -9711.45,E2 -9711.45} C_VEL
LIN {X 0,Y 425.546,Z 471.472,A -85,B 0,C 180,E1 -9714.313,E2 -9714.313} C_VEL
LIN {X 0,Y 425.566,Z 471.464,A -85,B 0,C 180,E1 -9718.107,E2 -9718.107} C_VEL
LIN {X 0,Y 425.695,Z 471.454,A -85,B 0,C 180,E1 -9720,E2 -9720} C_VEL
LIN {X 0,Y 425.549,Z 471.469,A -85,B 0,C 180,E1 -9722.84,E2 -9722.84} C_VEL
LIN {X 0,Y 425.569,Z 471.471,A -85,B 0,C 180,E1 -9725.687,E2 -9725.687} C_VEL
LIN {X 0,Y 425.433,Z 471.486,A -85,B 0,C 180,E1 -9728.55,E2 -9728.55} C_VEL
LIN {X 0,Y 425.403,Z 471.488,A -85,B 0,C 180,E1 -9732.402,E2 -9732.402} C_VEL
LIN {X 0,Y 425.379,Z 471.489,A -85,B 0,C 180,E1 -9736.312,E2 -9736.312} C_VEL
LIN {X 0,Y 425.32,Z 471.488,A -85,B 0,C 180,E1 -9739.636,E2 -9739.636} C_VEL
LIN {X 0,Y 425.299,Z 471.509,A -85,B 0,C 180,E1 -9743.366,E2 -9743.366} C_VEL
LIN {X 0,Y 425.341,Z 471.485,A -85,B 0,C 180,E1 -9746.845,E2 -9746.845} C_VEL
LIN {X 0,Y 425.312,Z 471.509,A -85,B 0,C 180,E1 -9749.718,E2 -9749.718} C_VEL
LIN {X 0,Y 425.278,Z 471.5,A -85,B 0,C 180,E1 -9753.048,E2 -9753.048} C_VEL
LIN {X 0,Y 425.279,Z 471.512,A -85,B 0,C 180,E1 -9755.93,E2 -9755.93} C_VEL
LIN {X 0,Y 425.298,Z 471.501,A -85,B 0,C 180,E1 -9759.045,E2 -9759.045} C_VEL
LIN {X 0,Y 425.27,Z 471.498,A -85,B 0,C 180,E1 -9762.654,E2 -9762.654} C_VEL
LIN {X 0,Y 425.331,Z 471.502,A -85,B 0,C 180,E1 -9766.054,E2 -9766.054} C_VEL
LIN {X 0,Y 425.306,Z 471.498,A -85,B 0,C 180,E1 -9768.626,E2 -9768.626} C_VEL
LIN {X 0,Y 425.319,Z 471.503,A -85,B 0,C 180,E1 -9771.105,E2 -9771.105} C_VEL
LIN {X 0,Y 425.298,Z 471.507,A -85,B 0,C 180,E1 -9774.665,E2 -9774.665} C_VEL
LIN {X 0,Y 425.335,Z 471.693,A -85,B 0,C 180,E1 -9777.997,E2 -9777.997} C_VEL
LIN {X 0,Y 428.783,Z 486.522,A -85,B 0,C 180,E1 -9780.547,E2 -9780.547} C_VEL
LIN {X 0,Y 430.047,Z 493.655,A -85,B 0,C 180,E1 -9781.711,E2 -9781.711} C_VEL
LIN {X 0,Y 428.784,Z 514.383,A -85,B 0,C 180,E1 -9784.777,E2 -9784.777} C_VEL
LIN {X 0,Y 427.508,Z 536.651,A -85,B 0,C 180,E1 -9788.038,E2 -9788.038} C_VEL
LIN {X 0,Y 426.498,Z 558.292,A -85,B 0,C 180,E1 -9791.199,E2 -9791.199} C_VEL
LIN {X 0,Y 430.134,Z 592.111,A -85,B 0,C 180,E1 -9791.96,E2 -9791.96} C_VEL
LIN {X 0,Y 429.407,Z 668.907,A -85,B 0,C 180,E1 -9793.265,E2 -9793.265} C_VEL
LIN {X 0,Y 428.819,Z 682.209,A -85,B 0,C 180,E1 -9793.67,E2 -9793.67} C_VEL
LIN {X 0,Y 428.153,Z 694.437,A -85,B 0,C 180,E1 -9794.225,E2 -9794.225} C_VEL
LIN {X 0,Y 427.434,Z 706.822,A -85,B 0,C 180,E1 -9794.992,E2 -9794.992} C_VEL
LIN {X 0,Y 426.663,Z 718.55,A -85,B 0,C 180,E1 -9795.939,E2 -9795.939} C_VEL
LIN {X 0,Y 426.023,Z 729.231,A -85,B 0,C 180,E1 -9797.02,E2 -9797.02} C_VEL
LIN {X 0,Y 425.403,Z 737.828,A -85,B 0,C 180,E1 -9798.082,E2 -9798.082} C_VEL
LIN {X 0,Y 425.021,Z 745.881,A -85,B 0,C 180,E1 -9799.279,E2 -9799.279} C_VEL
LIN {X 0,Y 424.724,Z 753.776,A -85,B 0,C 180,E1 -9800.716,E2 -9800.716} C_VEL
LIN {X 0,Y 424.557,Z 761.076,A -85,B 0,C 180,E1 -9802.39,E2 -9802.39} C_VEL
LIN {X 0,Y 424.559,Z 765.381,A -85,B 0,C 180,E1 -9803.637,E2 -9803.637} C_VEL
LIN {X 0,Y 424.669,Z 769.705,A -85,B 0,C 180,E1 -9805.254,E2 -9805.254} C_VEL
LIN {X 0,Y 424.713,Z 771.638,A -85,B 0,C 180,E1 -9806.205,E2 -9806.205} C_VEL
LIN {X 0,Y 424.693,Z 773.08,A -85,B 0,C 180,E1 -9807.154,E2 -9807.154} C_VEL
LIN {X 0,Y 424.933,Z 774.774,A -85,B 0,C 180,E1 -9809.052,E2 -9809.052} C_VEL
LIN {X 0,Y 424.945,Z 774.999,A -85,B 0,C 180,E1 -9810,E2 -9810} C_VEL
LIN {X 0,Y 424.933,Z 774.773,A -85,B 0,C 180,E1 -9810.948,E2 -9810.948} C_VEL
LIN {X 0,Y 424.693,Z 773.081,A -85,B 0,C 180,E1 -9812.846,E2 -9812.846} C_VEL
LIN {X 0,Y 424.713,Z 771.638,A -85,B 0,C 180,E1 -9813.795,E2 -9813.795} C_VEL
LIN {X 0,Y 424.611,Z 768.586,A -85,B 0,C 180,E1 -9815.223,E2 -9815.223} C_VEL
LIN {X 0,Y 424.541,Z 764.467,A -85,B 0,C 180,E1 -9816.654,E2 -9816.654} C_VEL
LIN {X 0,Y 424.611,Z 758.161,A -85,B 0,C 180,E1 -9818.327,E2 -9818.327} C_VEL
LIN {X 0,Y 424.799,Z 751.298,A -85,B 0,C 180,E1 -9819.763,E2 -9819.763} C_VEL
LIN {X 0,Y 425.189,Z 742.822,A -85,B 0,C 180,E1 -9821.199,E2 -9821.199} C_VEL
LIN {X 0,Y 425.741,Z 734.169,A -85,B 0,C 180,E1 -9822.392,E2 -9822.392} C_VEL
LIN {X 0,Y 426.308,Z 723.492,A -85,B 0,C 180,E1 -9823.587,E2 -9823.587} C_VEL
LIN {X 0,Y 427.038,Z 711.527,A -85,B 0,C 180,E1 -9824.657,E2 -9824.657} C_VEL
LIN {X 0,Y 427.865,Z 699.542,A -85,B 0,C 180,E1 -9825.481,E2 -9825.481} C_VEL
LIN {X 0,Y 428.573,Z 687.102,A -85,B 0,C 180,E1 -9826.126,E2 -9826.126} C_VEL
LIN {X 0,Y 429.221,Z 674.365,A -85,B 0,C 180,E1 -9826.589,E2 -9826.589} C_VEL
LIN {X 0,Y 429.519,Z 661.037,A -85,B 0,C 180,E1 -9826.884,E2 -9826.884} C_VEL
LIN {X 0,Y 430.047,Z 591.341,A -85,B 0,C 180,E1 -9828.052,E2 -9828.052} C_VEL
LIN {X 0,Y 426.483,Z 558.303,A -85,B 0,C 180,E1 -9828.796,E2 -9828.796} C_VEL
LIN {X 0,Y 427.618,Z 534.9,A -85,B 0,C 180,E1 -9832.21,E2 -9832.21} C_VEL
LIN {X 0,Y 428.986,Z 511.08,A -85,B 0,C 180,E1 -9835.702,E2 -9835.702} C_VEL
LIN {X 0,Y 430.043,Z 493.605,A -85,B 0,C 180,E1 -9838.289,E2 -9838.289} C_VEL
LIN {X 0,Y 428.578,Z 485.292,A -85,B 0,C 180,E1 -9839.644,E2 -9839.644} C_VEL
LIN {X 0,Y 425.316,Z 471.624,A -85,B 0,C 180,E1 -9842.032,E2 -9842.032} C_VEL
LIN {X 0,Y 425.297,Z 471.508,A -85,B 0,C 180,E1 -9845.335,E2 -9845.335} C_VEL
LIN {X 0,Y 425.308,Z 471.503,A -85,B 0,C 180,E1 -9849.045,E2 -9849.045} C_VEL
LIN {X 0,Y 425.328,Z 471.506,A -85,B 0,C 180,E1 -9852.645,E2 -9852.645} C_VEL
LIN {X 0,Y 425.29,Z 471.491,A -85,B 0,C 180,E1 -9855.281,E2 -9855.281} C_VEL
LIN {X 0,Y 425.27,Z 471.512,A -85,B 0,C 180,E1 -9858.621,E2 -9858.621} C_VEL
LIN {X 0,Y 425.31,Z 471.499,A -85,B 0,C 180,E1 -9861.102,E2 -9861.102} C_VEL
LIN {X 0,Y 425.294,Z 471.506,A -85,B 0,C 180,E1 -9864.664,E2 -9864.664} C_VEL
LIN {X 0,Y 425.261,Z 471.506,A -85,B 0,C 180,E1 -9868.073,E2 -9868.073} C_VEL
LIN {X 0,Y 425.331,Z 471.497,A -85,B 0,C 180,E1 -9871.368,E2 -9871.368} C_VEL
LIN {X 0,Y 425.288,Z 471.503,A -85,B 0,C 180,E1 -9874.554,E2 -9874.554} C_VEL
LIN {X 0,Y 425.28,Z 471.507,A -85,B 0,C 180,E1 -9877.661,E2 -9877.661} C_VEL
LIN {X 0,Y 425.353,Z 471.481,A -85,B 0,C 180,E1 -9880.704,E2 -9880.704} C_VEL
LIN {X 0,Y 425.38,Z 471.49,A -85,B 0,C 180,E1 -9883.688,E2 -9883.688} C_VEL
LIN {X 0,Y 425.403,Z 471.488,A -85,B 0,C 180,E1 -9887.598,E2 -9887.598} C_VEL
LIN {X 0,Y 425.434,Z 471.487,A -85,B 0,C 180,E1 -9891.45,E2 -9891.45} C_VEL
LIN {X 0,Y 425.569,Z 471.472,A -85,B 0,C 180,E1 -9894.313,E2 -9894.313} C_VEL
LIN {X 0,Y 425.567,Z 471.471,A -85,B 0,C 180,E1 -9898.107,E2 -9898.107} C_VEL
LIN {X 0,Y 425.695,Z 471.456,A -85,B 0,C 180,E1 -9900,E2 -9900} C_VEL
LIN {X 0,Y 425.549,Z 471.468,A -85,B 0,C 180,E1 -9902.84,E2 -9902.84} C_VEL
LIN {X 0,Y 425.57,Z 471.47,A -85,B 0,C 180,E1 -9905.687,E2 -9905.687} C_VEL
LIN {X 0,Y 425.434,Z 471.485,A -85,B 0,C 180,E1 -9908.55,E2 -9908.55} C_VEL
LIN {X 0,Y 425.403,Z 471.494,A -85,B 0,C 180,E1 -9912.402,E2 -9912.402} C_VEL
LIN {X 0,Y 425.38,Z 471.488,A -85,B 0,C 180,E1 -9916.312,E2 -9916.312} C_VEL
LIN {X 0,Y 425.32,Z 471.502,A -85,B 0,C 180,E1 -9919.636,E2 -9919.636} C_VEL
LIN {X 0,Y 425.299,Z 471.503,A -85,B 0,C 180,E1 -9923.366,E2 -9923.366} C_VEL
LIN {X 0,Y 425.344,Z 471.499,A -85,B 0,C 180,E1 -9926.846,E2 -9926.846} C_VEL
LIN {X 0,Y 425.311,Z 471.48,A -85,B 0,C 180,E1 -9929.718,E2 -9929.718} C_VEL
LIN {X 0,Y 425.276,Z 471.499,A -85,B 0,C 180,E1 -9933.049,E2 -9933.049} C_VEL
LIN {X 0,Y 425.279,Z 471.507,A -85,B 0,C 180,E1 -9935.93,E2 -9935.93} C_VEL
LIN {X 0,Y 425.279,Z 471.49,A -85,B 0,C 180,E1 -9939.042,E2 -9939.042} C_VEL
LIN {X 0,Y 425.286,Z 471.5,A -85,B 0,C 180,E1 -9941.959,E2 -9941.959} C_VEL
LIN {X 0,Y 425.285,Z 471.504,A -85,B 0,C 180,E1 -9945.283,E2 -9945.283} C_VEL
LIN {X 0,Y 425.273,Z 471.5,A -85,B 0,C 180,E1 -9948.622,E2 -9948.622} C_VEL
LIN {X 0,Y 425.315,Z 471.506,A -85,B 0,C 180,E1 -9951.104,E2 -9951.104} C_VEL
LIN {X 0,Y 425.299,Z 471.469,A -85,B 0,C 180,E1 -9954.665,E2 -9954.665} C_VEL
LIN {X 0,Y 425.265,Z 471.506,A -85,B 0,C 180,E1 -9958.074,E2 -9958.074} C_VEL
LIN {X 0,Y 425.331,Z 471.492,A -85,B 0,C 180,E1 -9961.369,E2 -9961.369} C_VEL
LIN {X 0,Y 425.296,Z 471.501,A -85,B 0,C 180,E1 -9964.555,E2 -9964.555} C_VEL
LIN {X 0,Y 425.289,Z 471.491,A -85,B 0,C 180,E1 -9967.662,E2 -9967.662} C_VEL
LIN {X 0,Y 425.354,Z 471.463,A -85,B 0,C 180,E1 -9971.205,E2 -9971.205} C_VEL
LIN {X 0,Y 425.409,Z 471.736,A -85,B 0,C 180,E1 -9971.582,E2 -9971.582} C_VEL
LIN {X 0,Y 425.669,Z 472.81,A -85,B 0,C 180,E1 -9971.718,E2 -9971.718} C_VEL
LIN {X 0,Y 430.881,Z 486.175,A -85,B 0,C 180,E1 -9972.202,E2 -9972.202} C_VEL
LIN {X 0,Y 430.467,Z 552.314,A -85,B 0,C 180,E1 -9973.338,E2 -9973.338} C_VEL
LIN {X 0,Y 430.351,Z 565.013,A -85,B 0,C 180,E1 -9973.73,E2 -9973.73} C_VEL
LIN {X 0,Y 430.036,Z 577.379,A -85,B 0,C 180,E1 -9974.296,E2 -9974.296} C_VEL
LIN {X 0,Y 429.644,Z 589.726,A -85,B 0,C 180,E1 -9975.069,E2 -9975.069} C_VEL
LIN {X 0,Y 428.968,Z 601.311,A -85,B 0,C 180,E1 -9976.016,E2 -9976.016} C_VEL
LIN {X 0,Y 428.352,Z 611.648,A -85,B 0,C 180,E1 -9977.083,E2 -9977.083} C_VEL
LIN {X 0,Y 427.797,Z 620.08,A -85,B 0,C 180,E1 -9978.15,E2 -9978.15} C_VEL
LIN {X 0,Y 427.317,Z 627.823,A -85,B 0,C 180,E1 -9979.338,E2 -9979.338} C_VEL
LIN {X 0,Y 426.703,Z 635.509,A -85,B 0,C 180,E1 -9980.783,E2 -9980.783} C_VEL
LIN {X 0,Y 426.315,Z 640.482,A -85,B 0,C 180,E1 -9981.932,E2 -9981.932} C_VEL
LIN {X 0,Y 425.516,Z 643.231,A -85,B 0,C 180,E1 -9982.63,E2 -9982.63} C_VEL
LIN {X 0,Y 422.374,Z 647.37,A -85,B 0,C 180,E1 -9983.771,E2 -9983.771} C_VEL
LIN {X 0,Y 419.212,Z 650.893,A -85,B 0,C 180,E1 -9984.962,E2 -9984.962} C_VEL
LIN {X 0,Y 418.398,Z 652.498,A -85,B 0,C 180,E1 -9985.73,E2 -9985.73} C_VEL
LIN {X 0,Y 418.359,Z 654.642,A -85,B 0,C 180,E1 -9987.111,E2 -9987.111} C_VEL
LIN {X 0,Y 418.203,Z 655.627,A -85,B 0,C 180,E1 -9988.074,E2 -9988.074} C_VEL
LIN {X 0,Y 418.28,Z 656.21,A -85,B 0,C 180,E1 -9989.037,E2 -9989.037} C_VEL
LIN {X 0,Y 418.263,Z 656.44,A -85,B 0,C 180,E1 -9990,E2 -9990} C_VEL
LIN {X 0,Y 418.28,Z 656.256,A -85,B 0,C 180,E1 -9990.963,E2 -9990.963} C_VEL
LIN {X 0,Y 418.203,Z 655.702,A -85,B 0,C 180,E1 -9991.926,E2 -9991.926} C_VEL
LIN {X 0,Y 418.357,Z 654.747,A -85,B 0,C 180,E1 -9992.889,E2 -9992.889} C_VEL
LIN {X 0,Y 418.333,Z 653.441,A -85,B 0,C 180,E1 -9993.853,E2 -9993.853} C_VEL
LIN {X 0,Y 418.614,Z 650.631,A -85,B 0,C 180,E1 -9995.298,E2 -9995.298} C_VEL
LIN {X 0,Y 419.043,Z 646.809,A -85,B 0,C 180,E1 -9996.742,E2 -9996.742} C_VEL
LIN {X 0,Y 419.32,Z 641.735,A -85,B 0,C 180,E1 -9998.239,E2 -9998.239} C_VEL
LIN {X 0,Y 419.84,Z 635.712,A -85,B 0,C 180,E1 -9999.636,E2 -9999.636} C_VEL
LIN {X 0,Y 420.507,Z 627.936,A -85,B 0,C 180,E1 -10001.081,E2 -10001.081} C_VEL
LIN {X 0,Y 421.14,Z 618.27,A -85,B 0,C 180,E1 -10002.529,E2 -10002.529} C_VEL
LIN {X 0,Y 421.778,Z 609.236,A -85,B 0,C 180,E1 -10003.613,E2 -10003.613} C_VEL
LIN {X 0,Y 422.464,Z 598.742,A -85,B 0,C 180,E1 -10004.628,E2 -10004.628} C_VEL
LIN {X 0,Y 422.956,Z 587.244,A -85,B 0,C 180,E1 -10005.518,E2 -10005.518} C_VEL
LIN {X 0,Y 423.392,Z 575.995,A -85,B 0,C 180,E1 -10006.186,E2 -10006.186} C_VEL
LIN {X 0,Y 423.692,Z 563.708,A -85,B 0,C 180,E1 -10006.719,E2 -10006.719} C_VEL
LIN {X 0,Y 423.722,Z 552.046,A -85,B 0,C 180,E1 -10007.059,E2 -10007.059} C_VEL
LIN {X 0,Y 424.142,Z 487.842,A -85,B 0,C 180,E1 -10008.177,E2 -10008.177} C_VEL
LIN {X 0,Y 418.508,Z 473.309,A -85,B 0,C 180,E1 -10008.73,E2 -10008.73} C_VEL
LIN {X 0,Y 418.339,Z 472.439,A -85,B 0,C 180,E1 -10008.932,E2 -10008.932} C_VEL
LIN {X 0,Y 418.239,Z 472.37,A -85,B 0,C 180,E1 -10012.735,E2 -10012.735} C_VEL
LIN {X 0,Y 418.271,Z 472.37,A -85,B 0,C 180,E1 -10015.903,E2 -10015.903} C_VEL
LIN {X 0,Y 418.265,Z 472.376,A -85,B 0,C 180,E1 -10019.161,E2 -10019.161} C_VEL
LIN {X 0,Y 418.257,Z 472.378,A -85,B 0,C 180,E1 -10022.843,E2 -10022.843} C_VEL
LIN {X 0,Y 418.247,Z 472.379,A -85,B 0,C 180,E1 -10026.238,E2 -10026.238} C_VEL
LIN {X 0,Y 418.25,Z 472.385,A -85,B 0,C 180,E1 -10029.681,E2 -10029.681} C_VEL
LIN {X 0,Y 418.229,Z 472.375,A -85,B 0,C 180,E1 -10032.321,E2 -10032.321} C_VEL
LIN {X 0,Y 418.234,Z 472.388,A -85,B 0,C 180,E1 -10035.108,E2 -10035.108} C_VEL
LIN {X 0,Y 418.236,Z 472.38,A -85,B 0,C 180,E1 -10037.766,E2 -10037.766} C_VEL
LIN {X 0,Y 418.246,Z 472.375,A -85,B 0,C 180,E1 -10041.557,E2 -10041.557} C_VEL
LIN {X 0,Y 418.254,Z 472.386,A -85,B 0,C 180,E1 -10045.158,E2 -10045.158} C_VEL
LIN {X 0,Y 418.24,Z 472.368,A -85,B 0,C 180,E1 -10047.471,E2 -10047.471} C_VEL
LIN {X 0,Y 418.27,Z 472.36,A -85,B 0,C 180,E1 -10050.893,E2 -10050.893} C_VEL
LIN {X 0,Y 418.264,Z 472.381,A -85,B 0,C 180,E1 -10054.095,E2 -10054.095} C_VEL
LIN {X 0,Y 418.23,Z 472.382,A -85,B 0,C 180,E1 -10057.263,E2 -10057.263} C_VEL
LIN {X 0,Y 418.275,Z 472.379,A -85,B 0,C 180,E1 -10060.364,E2 -10060.364} C_VEL
LIN {X 0,Y 418.308,Z 472.37,A -85,B 0,C 180,E1 -10063.404,E2 -10063.404} C_VEL
LIN {X 0,Y 418.338,Z 472.374,A -85,B 0,C 180,E1 -10066.999,E2 -10066.999} C_VEL
LIN {X 0,Y 418.333,Z 472.361,A -85,B 0,C 180,E1 -10070.328,E2 -10070.328} C_VEL
LIN {X 0,Y 418.504,Z 472.347,A -85,B 0,C 180,E1 -10072.279,E2 -10072.279} C_VEL
LIN {X 0,Y 418.505,Z 472.349,A -85,B 0,C 180,E1 -10074.217,E2 -10074.217} C_VEL
